LIN {X 0,Y 573.241,Z 599.114,A -85,B 0,C 180,E1 -2241.185,E2 -2241.185} C_VEL
LIN {X 0,Y 573.161,Z 606.962,A -85,B 0,C 180,E1 -2242.071,E2 -2242.071} C_VEL
LIN {X 0,Y 573.072,Z 614.955,A -85,B 0,C 180,E1 -2243.185,E2 -2243.185} C_VEL
LIN {X 0,Y 573.07,Z 621.68,A -85,B 0,C 180,E1 -2244.37,E2 -2244.37} C_VEL
LIN {X 0,Y 573.029,Z 626.372,A -85,B 0,C 180,E1 -2245.428,E2 -2245.428} C_VEL
LIN {X 0,Y 573.022,Z 629.957,A -85,B 0,C 180,E1 -2246.484,E2 -2246.484} C_VEL
LIN {X 0,Y 572.959,Z 631.808,A -85,B 0,C 180,E1 -2247.188,E2 -2247.188} C_VEL
LIN {X 0,Y 572.938,Z 633.198,A -85,B 0,C 180,E1 -2247.891,E2 -2247.891} C_VEL
LIN {X 0,Y 572.941,Z 634.785,A -85,B 0,C 180,E1 -2249.297,E2 -2249.297} C_VEL
LIN {X 0,Y 572.938,Z 635,A -85,B 0,C 180,E1 -2250,E2 -2250} C_VEL
LIN {X 0,Y 572.946,Z 634.186,A -85,B 0,C 180,E1 -2251.406,E2 -2251.406} C_VEL
LIN {X 0,Y 572.938,Z 633.2,A -85,B 0,C 180,E1 -2252.109,E2 -2252.109} C_VEL
LIN {X 0,Y 572.959,Z 631.81,A -85,B 0,C 180,E1 -2252.812,E2 -2252.812} C_VEL
LIN {X 0,Y 573.014,Z 628.896,A -85,B 0,C 180,E1 -2253.868,E2 -2253.868} C_VEL
LIN {X 0,Y 572.963,Z 624.949,A -85,B 0,C 180,E1 -2254.926,E2 -2254.926} C_VEL
LIN {X 0,Y 573.064,Z 618.877,A -85,B 0,C 180,E1 -2256.16,E2 -2256.16} C_VEL
LIN {X 0,Y 573.119,Z 612.238,A -85,B 0,C 180,E1 -2257.221,E2 -2257.221} C_VEL
LIN {X 0,Y 573.201,Z 603.992,A -85,B 0,C 180,E1 -2258.283,E2 -2258.283} C_VEL
LIN {X 0,Y 573.286,Z 595.54,A -85,B 0,C 180,E1 -2259.17,E2 -2259.17} C_VEL
LIN {X 0,Y 573.421,Z 585.101,A -85,B 0,C 180,E1 -2260.058,E2 -2260.058} C_VEL
LIN {X 0,Y 573.55,Z 573.355,A -85,B 0,C 180,E1 -2260.858,E2 -2260.858} C_VEL
LIN {X 0,Y 573.653,Z 562.287,A -85,B 0,C 180,E1 -2261.447,E2 -2261.447} C_VEL
LIN {X 0,Y 573.748,Z 549.178,A -85,B 0,C 180,E1 -2261.974,E2 -2261.974} C_VEL
LIN {X 0,Y 573.828,Z 536.528,A -85,B 0,C 180,E1 -2262.331,E2 -2262.331} C_VEL
LIN {X 0,Y 573.892,Z 523.328,A -85,B 0,C 180,E1 -2262.554,E2 -2262.554} C_VEL
LIN {X 0,Y 573.889,Z 423.833,A -85,B 0,C 180,E1 -2263.807,E2 -2263.807} C_VEL
LIN {X 0,Y 573.519,Z 420.897,A -85,B 0,C 180,E1 -2263.87,E2 -2263.87} C_VEL
LIN {X 0,Y 573.775,Z 395.95,A -85,B 0,C 180,E1 -2266.546,E2 -2266.546} C_VEL
LIN {X 0,Y 574.061,Z 369.009,A -85,B 0,C 180,E1 -2269.493,E2 -2269.493} C_VEL
LIN {X 0,Y 574.387,Z 343.84,A -85,B 0,C 180,E1 -2272.29,E2 -2272.29} C_VEL
LIN {X 0,Y 574.532,Z 322.946,A -85,B 0,C 180,E1 -2274.576,E2 -2274.576} C_VEL
LIN {X 0,Y 574.612,Z 306.194,A -85,B 0,C 180,E1 -2276.412,E2 -2276.412} C_VEL
LIN {X 0,Y 573.247,Z 300.208,A -85,B 0,C 180,E1 -2277.16,E2 -2277.16} C_VEL
LIN {X 0,Y 573.225,Z 300.08,A -85,B 0,C 180,E1 -2280.177,E2 -2280.177} C_VEL
LIN {X 0,Y 573.221,Z 300.078,A -85,B 0,C 180,E1 -2282.646,E2 -2282.646} C_VEL
LIN {X 0,Y 573.184,Z 300.082,A -85,B 0,C 180,E1 -2285.189,E2 -2285.189} C_VEL
LIN {X 0,Y 573.216,Z 300.084,A -85,B 0,C 180,E1 -2287.808,E2 -2287.808} C_VEL
LIN {X 0,Y 573.242,Z 300.076,A -85,B 0,C 180,E1 -2290.524,E2 -2290.524} C_VEL
LIN {X 0,Y 573.199,Z 300.084,A -85,B 0,C 180,E1 -2293.664,E2 -2293.664} C_VEL
LIN {X 0,Y 573.195,Z 300.08,A -85,B 0,C 180,E1 -2296.637,E2 -2296.637} C_VEL
LIN {X 0,Y 573.24,Z 300.077,A -85,B 0,C 180,E1 -2299.474,E2 -2299.474} C_VEL
LIN {X 0,Y 573.212,Z 300.075,A -85,B 0,C 180,E1 -2302.19,E2 -2302.19} C_VEL
LIN {X 0,Y 573.213,Z 300.075,A -85,B 0,C 180,E1 -2305.23,E2 -2305.23} C_VEL
LIN {X 0,Y 573.241,Z 300.082,A -85,B 0,C 180,E1 -2307.772,E2 -2307.772} C_VEL
LIN {X 0,Y 573.253,Z 300.071,A -85,B 0,C 180,E1 -2310.633,E2 -2310.633} C_VEL
LIN {X 0,Y 573.198,Z 300.083,A -85,B 0,C 180,E1 -2313.513,E2 -2313.513} C_VEL
LIN {X 0,Y 573.21,Z 300.082,A -85,B 0,C 180,E1 -2316.134,E2 -2316.134} C_VEL
LIN {X 0,Y 573.239,Z 300.072,A -85,B 0,C 180,E1 -2319.173,E2 -2319.173} C_VEL
LIN {X 0,Y 573.199,Z 300.081,A -85,B 0,C 180,E1 -2321.41,E2 -2321.41} C_VEL
LIN {X 0,Y 573.227,Z 300.083,A -85,B 0,C 180,E1 -2323.621,E2 -2323.621} C_VEL
LIN {X 0,Y 573.253,Z 300.08,A -85,B 0,C 180,E1 -2325.806,E2 -2325.806} C_VEL
LIN {X 0,Y 573.254,Z 300.072,A -85,B 0,C 180,E1 -2328.745,E2 -2328.745} C_VEL
LIN {X 0,Y 573.231,Z 300.082,A -85,B 0,C 180,E1 -2331.54,E2 -2331.54} C_VEL
LIN {X 0,Y 573.224,Z 300.084,A -85,B 0,C 180,E1 -2333.665,E2 -2333.665} C_VEL
LIN {X 0,Y 573.203,Z 300.088,A -85,B 0,C 180,E1 -2335.781,E2 -2335.781} C_VEL
LIN {X 0,Y 573.287,Z 300.075,A -85,B 0,C 180,E1 -2337.892,E2 -2337.892} C_VEL
LIN {X 0,Y 573.298,Z 300.069,A -85,B 0,C 180,E1 -2340,E2 -2340} C_VEL
LIN {X 0,Y 573.272,Z 300.069,A -85,B 0,C 180,E1 -2342.811,E2 -2342.811} C_VEL
LIN {X 0,Y 573.268,Z 300.08,A -85,B 0,C 180,E1 -2345.628,E2 -2345.628} C_VEL
LIN {X 0,Y 573.233,Z 300.073,A -85,B 0,C 180,E1 -2348.46,E2 -2348.46} C_VEL
LIN {X 0,Y 573.263,Z 300.076,A -85,B 0,C 180,E1 -2351.312,E2 -2351.312} C_VEL
LIN {X 0,Y 573.248,Z 300.071,A -85,B 0,C 180,E1 -2354.415,E2 -2354.415} C_VEL
LIN {X 0,Y 573.228,Z 300.078,A -85,B 0,C 180,E1 -2357.113,E2 -2357.113} C_VEL
LIN {X 0,Y 573.221,Z 300.077,A -85,B 0,C 180,E1 -2360.078,E2 -2360.078} C_VEL
LIN {X 0,Y 573.21,Z 300.078,A -85,B 0,C 180,E1 -2362.339,E2 -2362.339} C_VEL
LIN {X 0,Y 573.188,Z 300.081,A -85,B 0,C 180,E1 -2364.345,E2 -2364.345} C_VEL
LIN {X 0,Y 572.549,Z 300.162,A -85,B 0,C 180,E1 -2364.932,E2 -2364.932} C_VEL
LIN {X 0,Y 569.716,Z 300.521,A -85,B 0,C 180,E1 -2365.883,E2 -2365.883} C_VEL
LIN {X 0,Y 567.297,Z 300.825,A -85,B 0,C 180,E1 -2366.649,E2 -2366.649} C_VEL
LIN {X 0,Y 566.241,Z 300.953,A -85,B 0,C 180,E1 -2367.24,E2 -2367.24} C_VEL
LIN {X 0,Y 566.147,Z 300.961,A -85,B 0,C 180,E1 -2367.441,E2 -2367.441} C_VEL
LIN {X 0,Y 566.16,Z 300.956,A -85,B 0,C 180,E1 -2369.771,E2 -2369.771} C_VEL
LIN {X 0,Y 566.184,Z 300.951,A -85,B 0,C 180,E1 -2372.428,E2 -2372.428} C_VEL
LIN {X 0,Y 566.159,Z 300.959,A -85,B 0,C 180,E1 -2374.988,E2 -2374.988} C_VEL
LIN {X 0,Y 566.182,Z 300.959,A -85,B 0,C 180,E1 -2377.462,E2 -2377.462} C_VEL
LIN {X 0,Y 566.188,Z 300.95,A -85,B 0,C 180,E1 -2380.201,E2 -2380.201} C_VEL
LIN {X 0,Y 566.175,Z 300.958,A -85,B 0,C 180,E1 -2383.057,E2 -2383.057} C_VEL
LIN {X 0,Y 566.149,Z 300.955,A -85,B 0,C 180,E1 -2386.054,E2 -2386.054} C_VEL
LIN {X 0,Y 566.149,Z 300.959,A -85,B 0,C 180,E1 -2388.859,E2 -2388.859} C_VEL
LIN {X 0,Y 566.195,Z 300.958,A -85,B 0,C 180,E1 -2391.444,E2 -2391.444} C_VEL
LIN {X 0,Y 566.139,Z 300.958,A -85,B 0,C 180,E1 -2394.307,E2 -2394.307} C_VEL
LIN {X 0,Y 566.165,Z 300.958,A -85,B 0,C 180,E1 -2396.895,E2 -2396.895} C_VEL
LIN {X 0,Y 566.158,Z 300.965,A -85,B 0,C 180,E1 -2399.407,E2 -2399.407} C_VEL
LIN {X 0,Y 566.151,Z 300.954,A -85,B 0,C 180,E1 -2401.855,E2 -2401.855} C_VEL
LIN {X 0,Y 566.169,Z 300.955,A -85,B 0,C 180,E1 -2404.249,E2 -2404.249} C_VEL
LIN {X 0,Y 566.159,Z 300.961,A -85,B 0,C 180,E1 -2407.368,E2 -2407.368} C_VEL
LIN {X 0,Y 566.199,Z 300.956,A -85,B 0,C 180,E1 -2409.663,E2 -2409.663} C_VEL
LIN {X 0,Y 566.196,Z 300.944,A -85,B 0,C 180,E1 -2412.897,E2 -2412.897} C_VEL
LIN {X 0,Y 566.221,Z 300.986,A -85,B 0,C 180,E1 -2416.222,E2 -2416.222} C_VEL
LIN {X 0,Y 566.335,Z 301.687,A -85,B 0,C 180,E1 -2416.374,E2 -2416.374} C_VEL
LIN {X 0,Y 567.038,Z 303.971,A -85,B 0,C 180,E1 -2416.453,E2 -2416.453} C_VEL
LIN {X 0,Y 566.993,Z 380.985,A -85,B 0,C 180,E1 -2417.45,E2 -2417.45} C_VEL
LIN {X 0,Y 566.878,Z 394.243,A -85,B 0,C 180,E1 -2417.765,E2 -2417.765} C_VEL
LIN {X 0,Y 566.749,Z 406.398,A -85,B 0,C 180,E1 -2418.194,E2 -2418.194} C_VEL
LIN {X 0,Y 566.633,Z 418.541,A -85,B 0,C 180,E1 -2418.775,E2 -2418.775} C_VEL
LIN {X 0,Y 566.473,Z 429.557,A -85,B 0,C 180,E1 -2419.456,E2 -2419.456} C_VEL
LIN {X 0,Y 566.326,Z 440.075,A -85,B 0,C 180,E1 -2420.266,E2 -2420.266} C_VEL
LIN {X 0,Y 566.221,Z 448.673,A -85,B 0,C 180,E1 -2421.075,E2 -2421.075} C_VEL
LIN {X 0,Y 566.113,Z 456.592,A -85,B 0,C 180,E1 -2421.972,E2 -2421.972} C_VEL
LIN {X 0,Y 566.05,Z 463.16,A -85,B 0,C 180,E1 -2422.868,E2 -2422.868} C_VEL
LIN {X 0,Y 566.003,Z 469.628,A -85,B 0,C 180,E1 -2423.942,E2 -2423.942} C_VEL
LIN {X 0,Y 565.878,Z 474.766,A -85,B 0,C 180,E1 -2425.013,E2 -2425.013} C_VEL
LIN {X 0,Y 565.926,Z 478.754,A -85,B 0,C 180,E1 -2426.084,E2 -2426.084} C_VEL
LIN {X 0,Y 565.877,Z 481.704,A -85,B 0,C 180,E1 -2427.153,E2 -2427.153} C_VEL
LIN {X 0,Y 565.84,Z 483.127,A -85,B 0,C 180,E1 -2427.865,E2 -2427.865} C_VEL
LIN {X 0,Y 565.841,Z 484.756,A -85,B 0,C 180,E1 -2429.288,E2 -2429.288} C_VEL
LIN {X 0,Y 565.839,Z 484.996,A -85,B 0,C 180,E1 -2430,E2 -2430} C_VEL
LIN {X 0,Y 565.841,Z 484.815,A -85,B 0,C 180,E1 -2430.712,E2 -2430.712} C_VEL
LIN {X 0,Y 565.841,Z 483.269,A -85,B 0,C 180,E1 -2432.135,E2 -2432.135} C_VEL
LIN {X 0,Y 565.878,Z 481.908,A -85,B 0,C 180,E1 -2432.847,E2 -2432.847} C_VEL
LIN {X 0,Y 565.927,Z 479.029,A -85,B 0,C 180,E1 -2433.916,E2 -2433.916} C_VEL
LIN {X 0,Y 565.878,Z 475.129,A -85,B 0,C 180,E1 -2434.987,E2 -2434.987} C_VEL
LIN {X 0,Y 565.99,Z 470.098,A -85,B 0,C 180,E1 -2436.059,E2 -2436.059} C_VEL
LIN {X 0,Y 566.031,Z 463.773,A -85,B 0,C 180,E1 -2437.132,E2 -2437.132} C_VEL
LIN {X 0,Y 566.128,Z 455.85,A -85,B 0,C 180,E1 -2438.208,E2 -2438.208} C_VEL
LIN {X 0,Y 566.249,Z 445.997,A -85,B 0,C 180,E1 -2439.285,E2 -2439.285} C_VEL
LIN {X 0,Y 566.425,Z 435.682,A -85,B 0,C 180,E1 -2440.184,E2 -2440.184} C_VEL
LIN {X 0,Y 566.581,Z 424.398,A -85,B 0,C 180,E1 -2440.971,E2 -2440.971} C_VEL
LIN {X 0,Y 566.679,Z 412.486,A -85,B 0,C 180,E1 -2441.626,E2 -2441.626} C_VEL
LIN {X 0,Y 566.819,Z 400.474,A -85,B 0,C 180,E1 -2442.123,E2 -2442.123} C_VEL
LIN {X 0,Y 566.928,Z 387.43,A -85,B 0,C 180,E1 -2442.506,E2 -2442.506} C_VEL
LIN {X 0,Y 567.026,Z 375.066,A -85,B 0,C 180,E1 -2442.732,E2 -2442.732} C_VEL
LIN {X 0,Y 567.08,Z 304.212,A -85,B 0,C 180,E1 -2443.633,E2 -2443.633} C_VEL
LIN {X 0,Y 566.353,Z 301.818,A -85,B 0,C 180,E1 -2443.706,E2 -2443.706} C_VEL
LIN {X 0,Y 566.205,Z 301.005,A -85,B 0,C 180,E1 -2443.847,E2 -2443.847} C_VEL
LIN {X 0,Y 566.195,Z 300.93,A -85,B 0,C 180,E1 -2447.102,E2 -2447.102} C_VEL
LIN {X 0,Y 566.172,Z 300.956,A -85,B 0,C 180,E1 -2449.582,E2 -2449.582} C_VEL
LIN {X 0,Y 566.181,Z 300.952,A -85,B 0,C 180,E1 -2451.863,E2 -2451.863} C_VEL
LIN {X 0,Y 566.146,Z 300.959,A -85,B 0,C 180,E1 -2454.183,E2 -2454.183} C_VEL
LIN {X 0,Y 566.162,Z 300.961,A -85,B 0,C 180,E1 -2456.649,E2 -2456.649} C_VEL
LIN {X 0,Y 566.154,Z 300.957,A -85,B 0,C 180,E1 -2459.771,E2 -2459.771} C_VEL
LIN {X 0,Y 566.175,Z 300.959,A -85,B 0,C 180,E1 -2462.425,E2 -2462.425} C_VEL
LIN {X 0,Y 566.165,Z 300.961,A -85,B 0,C 180,E1 -2464.987,E2 -2464.987} C_VEL
LIN {X 0,Y 566.18,Z 300.952,A -85,B 0,C 180,E1 -2467.461,E2 -2467.461} C_VEL
LIN {X 0,Y 566.2,Z 300.954,A -85,B 0,C 180,E1 -2470.199,E2 -2470.199} C_VEL
LIN {X 0,Y 566.142,Z 300.959,A -85,B 0,C 180,E1 -2473.059,E2 -2473.059} C_VEL
LIN {X 0,Y 566.14,Z 300.96,A -85,B 0,C 180,E1 -2476.054,E2 -2476.054} C_VEL
LIN {X 0,Y 566.156,Z 300.955,A -85,B 0,C 180,E1 -2479.219,E2 -2479.219} C_VEL
LIN {X 0,Y 566.164,Z 300.951,A -85,B 0,C 180,E1 -2481.635,E2 -2481.635} C_VEL
LIN {X 0,Y 566.132,Z 300.964,A -85,B 0,C 180,E1 -2484.305,E2 -2484.305} C_VEL
LIN {X 0,Y 566.187,Z 300.956,A -85,B 0,C 180,E1 -2486.895,E2 -2486.895} C_VEL
LIN {X 0,Y 566.146,Z 300.952,A -85,B 0,C 180,E1 -2489.405,E2 -2489.405} C_VEL
LIN {X 0,Y 566.139,Z 300.954,A -85,B 0,C 180,E1 -2491.853,E2 -2491.853} C_VEL
LIN {X 0,Y 566.184,Z 300.957,A -85,B 0,C 180,E1 -2494.249,E2 -2494.249} C_VEL
LIN {X 0,Y 566.13,Z 300.959,A -85,B 0,C 180,E1 -2497.366,E2 -2497.366} C_VEL
LIN {X 0,Y 566.161,Z 300.954,A -85,B 0,C 180,E1 -2499.661,E2 -2499.661} C_VEL
LIN {X 0,Y 566.161,Z 300.958,A -85,B 0,C 180,E1 -2501.92,E2 -2501.92} C_VEL
LIN {X 0,Y 566.17,Z 300.955,A -85,B 0,C 180,E1 -2504.89,E2 -2504.89} C_VEL
LIN {X 0,Y 566.163,Z 300.957,A -85,B 0,C 180,E1 -2507.817,E2 -2507.817} C_VEL
LIN {X 0,Y 566.143,Z 300.961,A -85,B 0,C 180,E1 -2509.991,E2 -2509.991} C_VEL
LIN {X 0,Y 566.176,Z 300.956,A -85,B 0,C 180,E1 -2512.869,E2 -2512.869} C_VEL
LIN {X 0,Y 566.245,Z 300.947,A -85,B 0,C 180,E1 -2515.016,E2 -2515.016} C_VEL
LIN {X 0,Y 566.254,Z 300.946,A -85,B 0,C 180,E1 -2517.866,E2 -2517.866} C_VEL
LIN {X 0,Y 566.289,Z 300.944,A -85,B 0,C 180,E1 -2520.711,E2 -2520.711} C_VEL
LIN {X 0,Y 566.247,Z 300.947,A -85,B 0,C 180,E1 -2522.846,E2 -2522.846} C_VEL
LIN {X 0,Y 566.224,Z 300.948,A -85,B 0,C 180,E1 -2525.699,E2 -2525.699} C_VEL
LIN {X 0,Y 566.174,Z 300.956,A -85,B 0,C 180,E1 -2527.848,E2 -2527.848} C_VEL
LIN {X 0,Y 566.204,Z 300.953,A -85,B 0,C 180,E1 -2530.73,E2 -2530.73} C_VEL
LIN {X 0,Y 566.171,Z 300.954,A -85,B 0,C 180,E1 -2533.642,E2 -2533.642} C_VEL
LIN {X 0,Y 566.175,Z 300.958,A -85,B 0,C 180,E1 -2535.848,E2 -2535.848} C_VEL
LIN {X 0,Y 566.18,Z 300.953,A -85,B 0,C 180,E1 -2538.829,E2 -2538.829} C_VEL
LIN {X 0,Y 566.2,Z 300.948,A -85,B 0,C 180,E1 -2541.42,E2 -2541.42} C_VEL
LIN {X 0,Y 566.163,Z 300.965,A -85,B 0,C 180,E1 -2544.182,E2 -2544.182} C_VEL
LIN {X 0,Y 566.166,Z 300.956,A -85,B 0,C 180,E1 -2546.653,E2 -2546.653} C_VEL
LIN {X 0,Y 566.166,Z 300.954,A -85,B 0,C 180,E1 -2548.955,E2 -2548.955} C_VEL
LIN {X 0,Y 566.182,Z 300.954,A -85,B 0,C 180,E1 -2551.423,E2 -2551.423} C_VEL
LIN {X 0,Y 566.188,Z 300.959,A -85,B 0,C 180,E1 -2553.958,E2 -2553.958} C_VEL
LIN {X 0,Y 566.138,Z 300.962,A -85,B 0,C 180,E1 -2556.575,E2 -2556.575} C_VEL
LIN {X 0,Y 566.2,Z 300.95,A -85,B 0,C 180,E1 -2559.275,E2 -2559.275} C_VEL
LIN {X 0,Y 566.173,Z 300.964,A -85,B 0,C 180,E1 -2562.091,E2 -2562.091} C_VEL
LIN {X 0,Y 566.159,Z 300.951,A -85,B 0,C 180,E1 -2565.038,E2 -2565.038} C_VEL
LIN {X 0,Y 566.158,Z 300.964,A -85,B 0,C 180,E1 -2568.143,E2 -2568.143} C_VEL
LIN {X 0,Y 566.204,Z 300.95,A -85,B 0,C 180,E1 -2570.726,E2 -2570.726} C_VEL
LIN {X 0,Y 566.139,Z 300.961,A -85,B 0,C 180,E1 -2573.426,E2 -2573.426} C_VEL
LIN {X 0,Y 566.193,Z 300.956,A -85,B 0,C 180,E1 -2576.269,E2 -2576.269} C_VEL
LIN {X 0,Y 566.181,Z 300.954,A -85,B 0,C 180,E1 -2578.926,E2 -2578.926} C_VEL
LIN {X 0,Y 566.147,Z 300.965,A -85,B 0,C 180,E1 -2581.854,E2 -2581.854} C_VEL
LIN {X 0,Y 566.189,Z 301.12,A -85,B 0,C 180,E1 -2582.681,E2 -2582.681} C_VEL
LIN {X 0,Y 567.751,Z 307.979,A -85,B 0,C 180,E1 -2583.537,E2 -2583.537} C_VEL
LIN {X 0,Y 567.58,Z 332.208,A -85,B 0,C 180,E1 -2586.22,E2 -2586.22} C_VEL
LIN {X 0,Y 567.362,Z 357.278,A -85,B 0,C 180,E1 -2588.948,E2 -2588.948} C_VEL
LIN {X 0,Y 566.967,Z 384.183,A -85,B 0,C 180,E1 -2591.947,E2 -2591.947} C_VEL
LIN {X 0,Y 566.677,Z 409.398,A -85,B 0,C 180,E1 -2594.72,E2 -2594.72} C_VEL
LIN {X 0,Y 566.563,Z 420.903,A -85,B 0,C 180,E1 -2595.956,E2 -2595.956} C_VEL
LIN {X 0,Y 567.197,Z 426.739,A -85,B 0,C 180,E1 -2596.064,E2 -2596.064} C_VEL
LIN {X 0,Y 566.97,Z 530.957,A -85,B 0,C 180,E1 -2597.404,E2 -2597.404} C_VEL
LIN {X 0,Y 566.892,Z 543.463,A -85,B 0,C 180,E1 -2597.697,E2 -2597.697} C_VEL
LIN {X 0,Y 566.747,Z 555.924,A -85,B 0,C 180,E1 -2598.13,E2 -2598.13} C_VEL
LIN {X 0,Y 566.627,Z 568.166,A -85,B 0,C 180,E1 -2598.709,E2 -2598.709} C_VEL
LIN {X 0,Y 566.457,Z 580.202,A -85,B 0,C 180,E1 -2599.456,E2 -2599.456} C_VEL
LIN {X 0,Y 566.321,Z 590.604,A -85,B 0,C 180,E1 -2600.266,E2 -2600.266} C_VEL
LIN {X 0,Y 566.207,Z 599.114,A -85,B 0,C 180,E1 -2601.074,E2 -2601.074} C_VEL
LIN {X 0,Y 566.112,Z 606.962,A -85,B 0,C 180,E1 -2601.972,E2 -2601.972} C_VEL
LIN {X 0,Y 566.003,Z 614.623,A -85,B 0,C 180,E1 -2603.047,E2 -2603.047} C_VEL
LIN {X 0,Y 566.004,Z 621.68,A -85,B 0,C 180,E1 -2604.299,E2 -2604.299} C_VEL
LIN {X 0,Y 565.933,Z 626.372,A -85,B 0,C 180,E1 -2605.37,E2 -2605.37} C_VEL
LIN {X 0,Y 565.927,Z 629.958,A -85,B 0,C 180,E1 -2606.44,E2 -2606.44} C_VEL
LIN {X 0,Y 565.878,Z 631.808,A -85,B 0,C 180,E1 -2607.152,E2 -2607.152} C_VEL
LIN {X 0,Y 565.846,Z 634.185,A -85,B 0,C 180,E1 -2608.577,E2 -2608.577} C_VEL
LIN {X 0,Y 565.839,Z 635,A -85,B 0,C 180,E1 -2610,E2 -2610} C_VEL
LIN {X 0,Y 565.846,Z 634.186,A -85,B 0,C 180,E1 -2611.423,E2 -2611.423} C_VEL
LIN {X 0,Y 565.878,Z 631.81,A -85,B 0,C 180,E1 -2612.847,E2 -2612.847} C_VEL
LIN {X 0,Y 565.926,Z 628.896,A -85,B 0,C 180,E1 -2613.916,E2 -2613.916} C_VEL
LIN {X 0,Y 565.878,Z 624.949,A -85,B 0,C 180,E1 -2614.987,E2 -2614.987} C_VEL
LIN {X 0,Y 566.002,Z 619.867,A -85,B 0,C 180,E1 -2616.058,E2 -2616.058} C_VEL
LIN {X 0,Y 566.04,Z 613.469,A -85,B 0,C 180,E1 -2617.132,E2 -2617.132} C_VEL
LIN {X 0,Y 566.133,Z 605.479,A -85,B 0,C 180,E1 -2618.208,E2 -2618.208} C_VEL
LIN {X 0,Y 566.228,Z 597.337,A -85,B 0,C 180,E1 -2619.105,E2 -2619.105} C_VEL
LIN {X 0,Y 566.342,Z 587.402,A -85,B 0,C 180,E1 -2620.005,E2 -2620.005} C_VEL
LIN {X 0,Y 566.525,Z 576.288,A -85,B 0,C 180,E1 -2620.808,E2 -2620.808} C_VEL
LIN {X 0,Y 566.66,Z 565.18,A -85,B 0,C 180,E1 -2621.446,E2 -2621.446} C_VEL
LIN {X 0,Y 566.737,Z 552.988,A -85,B 0,C 180,E1 -2621.988,E2 -2621.988} C_VEL
LIN {X 0,Y 566.906,Z 540.185,A -85,B 0,C 180,E1 -2622.393,E2 -2622.393} C_VEL
LIN {X 0,Y 566.995,Z 526.617,A -85,B 0,C 180,E1 -2622.664,E2 -2622.664} C_VEL
LIN {X 0,Y 567.067,Z 424.95,A -85,B 0,C 180,E1 -2623.962,E2 -2623.962} C_VEL
LIN {X 0,Y 566.562,Z 420.904,A -85,B 0,C 180,E1 -2624.044,E2 -2624.044} C_VEL
LIN {X 0,Y 566.844,Z 394.447,A -85,B 0,C 180,E1 -2626.92,E2 -2626.92} C_VEL
LIN {X 0,Y 567.215,Z 367.71,A -85,B 0,C 180,E1 -2629.884,E2 -2629.884} C_VEL
LIN {X 0,Y 567.445,Z 346.786,A -85,B 0,C 180,E1 -2632.194,E2 -2632.194} C_VEL
LIN {X 0,Y 567.647,Z 322.094,A -85,B 0,C 180,E1 -2634.894,E2 -2634.894} C_VEL
LIN {X 0,Y 567.737,Z 307.968,A -85,B 0,C 180,E1 -2636.464,E2 -2636.464} C_VEL
LIN {X 0,Y 566.207,Z 301.1,A -85,B 0,C 180,E1 -2637.32,E2 -2637.32} C_VEL
LIN {X 0,Y 566.158,Z 300.954,A -85,B 0,C 180,E1 -2639.771,E2 -2639.771} C_VEL
LIN {X 0,Y 566.176,Z 300.958,A -85,B 0,C 180,E1 -2642.425,E2 -2642.425} C_VEL
LIN {X 0,Y 566.16,Z 300.956,A -85,B 0,C 180,E1 -2644.986,E2 -2644.986} C_VEL
LIN {X 0,Y 566.182,Z 300.956,A -85,B 0,C 180,E1 -2647.461,E2 -2647.461} C_VEL
LIN {X 0,Y 566.202,Z 300.957,A -85,B 0,C 180,E1 -2650.199,E2 -2650.199} C_VEL
LIN {X 0,Y 566.143,Z 300.958,A -85,B 0,C 180,E1 -2653.059,E2 -2653.059} C_VEL
LIN {X 0,Y 566.152,Z 300.964,A -85,B 0,C 180,E1 -2656.053,E2 -2656.053} C_VEL
LIN {X 0,Y 566.151,Z 300.957,A -85,B 0,C 180,E1 -2658.858,E2 -2658.858} C_VEL
LIN {X 0,Y 566.195,Z 300.952,A -85,B 0,C 180,E1 -2661.443,E2 -2661.443} C_VEL
LIN {X 0,Y 566.133,Z 300.959,A -85,B 0,C 180,E1 -2664.306,E2 -2664.306} C_VEL
LIN {X 0,Y 566.191,Z 300.952,A -85,B 0,C 180,E1 -2666.896,E2 -2666.896} C_VEL
LIN {X 0,Y 566.174,Z 300.957,A -85,B 0,C 180,E1 -2669.407,E2 -2669.407} C_VEL
LIN {X 0,Y 566.18,Z 300.96,A -85,B 0,C 180,E1 -2671.856,E2 -2671.856} C_VEL
LIN {X 0,Y 566.179,Z 300.957,A -85,B 0,C 180,E1 -2674.249,E2 -2674.249} C_VEL
LIN {X 0,Y 566.157,Z 300.956,A -85,B 0,C 180,E1 -2676.72,E2 -2676.72} C_VEL
LIN {X 0,Y 566.195,Z 300.955,A -85,B 0,C 180,E1 -2679.662,E2 -2679.662} C_VEL
LIN {X 0,Y 566.169,Z 300.963,A -85,B 0,C 180,E1 -2681.921,E2 -2681.921} C_VEL
LIN {X 0,Y 566.18,Z 300.957,A -85,B 0,C 180,E1 -2684.152,E2 -2684.152} C_VEL
LIN {X 0,Y 566.171,Z 300.954,A -85,B 0,C 180,E1 -2686.358,E2 -2686.358} C_VEL
LIN {X 0,Y 566.222,Z 300.95,A -85,B 0,C 180,E1 -2689.27,E2 -2689.27} C_VEL
LIN {X 0,Y 566.175,Z 300.956,A -85,B 0,C 180,E1 -2692.152,E2 -2692.152} C_VEL
LIN {X 0,Y 566.226,Z 300.948,A -85,B 0,C 180,E1 -2694.301,E2 -2694.301} C_VEL
LIN {X 0,Y 566.248,Z 300.947,A -85,B 0,C 180,E1 -2697.154,E2 -2697.154} C_VEL
LIN {X 0,Y 566.268,Z 300.945,A -85,B 0,C 180,E1 -2700,E2 -2700} C_VEL
LIN {X 0,Y 566.242,Z 300.945,A -85,B 0,C 180,E1 -2702.846,E2 -2702.846} C_VEL
LIN {X 0,Y 566.235,Z 300.955,A -85,B 0,C 180,E1 -2705.699,E2 -2705.699} C_VEL
LIN {X 0,Y 566.185,Z 300.951,A -85,B 0,C 180,E1 -2708.566,E2 -2708.566} C_VEL
LIN {X 0,Y 566.23,Z 300.954,A -85,B 0,C 180,E1 -2711.455,E2 -2711.455} C_VEL
LIN {X 0,Y 566.204,Z 300.948,A -85,B 0,C 180,E1 -2714.498,E2 -2714.498} C_VEL
LIN {X 0,Y 566.173,Z 300.96,A -85,B 0,C 180,E1 -2717.333,E2 -2717.333} C_VEL
LIN {X 0,Y 566.19,Z 300.961,A -85,B 0,C 180,E1 -2719.582,E2 -2719.582} C_VEL
LIN {X 0,Y 566.176,Z 300.958,A -85,B 0,C 180,E1 -2721.863,E2 -2721.863} C_VEL
LIN {X 0,Y 566.17,Z 300.957,A -85,B 0,C 180,E1 -2725.022,E2 -2725.022} C_VEL
LIN {X 0,Y 566.147,Z 300.961,A -85,B 0,C 180,E1 -2727.441,E2 -2727.441} C_VEL
LIN {X 0,Y 565.459,Z 301.041,A -85,B 0,C 180,E1 -2728.034,E2 -2728.034} C_VEL
LIN {X 0,Y 562.605,Z 301.395,A -85,B 0,C 180,E1 -2728.999,E2 -2728.999} C_VEL
LIN {X 0,Y 560.214,Z 301.696,A -85,B 0,C 180,E1 -2729.775,E2 -2729.775} C_VEL
LIN {X 0,Y 559.197,Z 301.817,A -85,B 0,C 180,E1 -2730.373,E2 -2730.373} C_VEL
LIN {X 0,Y 559.118,Z 301.827,A -85,B 0,C 180,E1 -2730.576,E2 -2730.576} C_VEL
LIN {X 0,Y 559.14,Z 301.829,A -85,B 0,C 180,E1 -2732.717,E2 -2732.717} C_VEL
LIN {X 0,Y 559.109,Z 301.842,A -85,B 0,C 180,E1 -2735.326,E2 -2735.326} C_VEL
LIN {X 0,Y 559.116,Z 301.831,A -85,B 0,C 180,E1 -2738.019,E2 -2738.019} C_VEL
LIN {X 0,Y 559.143,Z 301.829,A -85,B 0,C 180,E1 -2739.941,E2 -2739.941} C_VEL
LIN {X 0,Y 559.12,Z 301.839,A -85,B 0,C 180,E1 -2743.195,E2 -2743.195} C_VEL
LIN {X 0,Y 559.116,Z 301.834,A -85,B 0,C 180,E1 -2745.765,E2 -2745.765} C_VEL
LIN {X 0,Y 559.096,Z 301.835,A -85,B 0,C 180,E1 -2748.225,E2 -2748.225} C_VEL
LIN {X 0,Y 559.163,Z 301.833,A -85,B 0,C 180,E1 -2751.066,E2 -2751.066} C_VEL
LIN {X 0,Y 559.113,Z 301.837,A -85,B 0,C 180,E1 -2753.788,E2 -2753.788} C_VEL
LIN {X 0,Y 559.123,Z 301.832,A -85,B 0,C 180,E1 -2756.423,E2 -2756.423} C_VEL
LIN {X 0,Y 559.142,Z 301.834,A -85,B 0,C 180,E1 -2758.98,E2 -2758.98} C_VEL
LIN {X 0,Y 559.111,Z 301.833,A -85,B 0,C 180,E1 -2761.63,E2 -2761.63} C_VEL
LIN {X 0,Y 559.14,Z 301.832,A -85,B 0,C 180,E1 -2763.901,E2 -2763.901} C_VEL
LIN {X 0,Y 559.11,Z 301.841,A -85,B 0,C 180,E1 -2767.067,E2 -2767.067} C_VEL
LIN {X 0,Y 559.171,Z 301.835,A -85,B 0,C 180,E1 -2769.396,E2 -2769.396} C_VEL
LIN {X 0,Y 559.122,Z 301.822,A -85,B 0,C 180,E1 -2772.442,E2 -2772.442} C_VEL
LIN {X 0,Y 559.154,Z 301.835,A -85,B 0,C 180,E1 -2775.441,E2 -2775.441} C_VEL
LIN {X 0,Y 559.229,Z 302.09,A -85,B 0,C 180,E1 -2776.14,E2 -2776.14} C_VEL
LIN {X 0,Y 559.536,Z 303.423,A -85,B 0,C 180,E1 -2776.248,E2 -2776.248} C_VEL
LIN {X 0,Y 560.273,Z 305.992,A -85,B 0,C 180,E1 -2776.305,E2 -2776.305} C_VEL
LIN {X 0,Y 560.089,Z 381.28,A -85,B 0,C 180,E1 -2777.292,E2 -2777.292} C_VEL
LIN {X 0,Y 559.939,Z 394.48,A -85,B 0,C 180,E1 -2777.611,E2 -2777.611} C_VEL
LIN {X 0,Y 559.798,Z 406.547,A -85,B 0,C 180,E1 -2778.045,E2 -2778.045} C_VEL
LIN {X 0,Y 559.648,Z 418.106,A -85,B 0,C 180,E1 -2778.607,E2 -2778.607} C_VEL
LIN {X 0,Y 559.489,Z 429.562,A -85,B 0,C 180,E1 -2779.323,E2 -2779.323} C_VEL
LIN {X 0,Y 559.307,Z 440.08,A -85,B 0,C 180,E1 -2780.142,E2 -2780.142} C_VEL
LIN {X 0,Y 559.197,Z 448.678,A -85,B 0,C 180,E1 -2780.962,E2 -2780.962} C_VEL
LIN {X 0,Y 559.05,Z 456.597,A -85,B 0,C 180,E1 -2781.87,E2 -2781.87} C_VEL
LIN {X 0,Y 558.971,Z 464.457,A -85,B 0,C 180,E1 -2782.977,E2 -2782.977} C_VEL
LIN {X 0,Y 558.936,Z 471.455,A -85,B 0,C 180,E1 -2784.227,E2 -2784.227} C_VEL
LIN {X 0,Y 558.827,Z 476.197,A -85,B 0,C 180,E1 -2785.311,E2 -2785.311} C_VEL
LIN {X 0,Y 558.836,Z 479.828,A -85,B 0,C 180,E1 -2786.395,E2 -2786.395} C_VEL
LIN {X 0,Y 558.799,Z 481.706,A -85,B 0,C 180,E1 -2787.116,E2 -2787.116} C_VEL
LIN {X 0,Y 558.746,Z 483.128,A -85,B 0,C 180,E1 -2787.838,E2 -2787.838} C_VEL
LIN {X 0,Y 558.741,Z 484.756,A -85,B 0,C 180,E1 -2789.279,E2 -2789.279} C_VEL
LIN {X 0,Y 558.74,Z 484.996,A -85,B 0,C 180,E1 -2790,E2 -2790} C_VEL
LIN {X 0,Y 558.741,Z 484.815,A -85,B 0,C 180,E1 -2790.721,E2 -2790.721} C_VEL
LIN {X 0,Y 558.746,Z 483.268,A -85,B 0,C 180,E1 -2792.163,E2 -2792.163} C_VEL
LIN {X 0,Y 558.8,Z 481.907,A -85,B 0,C 180,E1 -2792.884,E2 -2792.884} C_VEL
LIN {X 0,Y 558.844,Z 479.027,A -85,B 0,C 180,E1 -2793.966,E2 -2793.966} C_VEL
LIN {X 0,Y 558.798,Z 475.127,A -85,B 0,C 180,E1 -2795.051,E2 -2795.051} C_VEL
LIN {X 0,Y 558.91,Z 470.095,A -85,B 0,C 180,E1 -2796.136,E2 -2796.136} C_VEL
LIN {X 0,Y 558.972,Z 463.769,A -85,B 0,C 180,E1 -2797.223,E2 -2797.223} C_VEL
LIN {X 0,Y 559.091,Z 455.845,A -85,B 0,C 180,E1 -2798.312,E2 -2798.312} C_VEL
LIN {X 0,Y 559.182,Z 447.774,A -85,B 0,C 180,E1 -2799.221,E2 -2799.221} C_VEL
LIN {X 0,Y 559.357,Z 437.924,A -85,B 0,C 180,E1 -2800.131,E2 -2800.131} C_VEL
LIN {X 0,Y 559.581,Z 427.089,A -85,B 0,C 180,E1 -2800.937,E2 -2800.937} C_VEL
LIN {X 0,Y 559.68,Z 415.301,A -85,B 0,C 180,E1 -2801.631,E2 -2801.631} C_VEL
LIN {X 0,Y 559.832,Z 403.126,A -85,B 0,C 180,E1 -2802.184,E2 -2802.184} C_VEL
LIN {X 0,Y 559.976,Z 390.397,A -85,B 0,C 180,E1 -2802.595,E2 -2802.595} C_VEL
LIN {X 0,Y 560.135,Z 378.322,A -85,B 0,C 180,E1 -2802.845,E2 -2802.845} C_VEL
LIN {X 0,Y 560.265,Z 305.8,A -85,B 0,C 180,E1 -2803.788,E2 -2803.788} C_VEL
LIN {X 0,Y 559.318,Z 302.662,A -85,B 0,C 180,E1 -2803.88,E2 -2803.88} C_VEL
LIN {X 0,Y 559.165,Z 301.88,A -85,B 0,C 180,E1 -2804.021,E2 -2804.021} C_VEL
LIN {X 0,Y 559.149,Z 301.804,A -85,B 0,C 180,E1 -2807.204,E2 -2807.204} C_VEL
LIN {X 0,Y 559.138,Z 301.832,A -85,B 0,C 180,E1 -2809.838,E2 -2809.838} C_VEL
LIN {X 0,Y 559.125,Z 301.832,A -85,B 0,C 180,E1 -2812.153,E2 -2812.153} C_VEL
LIN {X 0,Y 559.115,Z 301.837,A -85,B 0,C 180,E1 -2815.172,E2 -2815.172} C_VEL
LIN {X 0,Y 559.102,Z 301.829,A -85,B 0,C 180,E1 -2817.716,E2 -2817.716} C_VEL
LIN {X 0,Y 559.098,Z 301.837,A -85,B 0,C 180,E1 -2820.185,E2 -2820.185} C_VEL
LIN {X 0,Y 559.133,Z 301.839,A -85,B 0,C 180,E1 -2822.716,E2 -2822.716} C_VEL
LIN {X 0,Y 559.115,Z 301.835,A -85,B 0,C 180,E1 -2825.324,E2 -2825.324} C_VEL
LIN {X 0,Y 559.117,Z 301.832,A -85,B 0,C 180,E1 -2828.018,E2 -2828.018} C_VEL
LIN {X 0,Y 559.12,Z 301.84,A -85,B 0,C 180,E1 -2830.815,E2 -2830.815} C_VEL
LIN {X 0,Y 559.094,Z 301.832,A -85,B 0,C 180,E1 -2833.738,E2 -2833.738} C_VEL
LIN {X 0,Y 559.088,Z 301.841,A -85,B 0,C 180,E1 -2836.261,E2 -2836.261} C_VEL
LIN {X 0,Y 559.109,Z 301.833,A -85,B 0,C 180,E1 -2839.183,E2 -2839.183} C_VEL
LIN {X 0,Y 559.137,Z 301.828,A -85,B 0,C 180,E1 -2841.195,E2 -2841.195} C_VEL
LIN {X 0,Y 559.109,Z 301.834,A -85,B 0,C 180,E1 -2843.787,E2 -2843.787} C_VEL
LIN {X 0,Y 559.138,Z 301.838,A -85,B 0,C 180,E1 -2846.423,E2 -2846.423} C_VEL
LIN {X 0,Y 559.133,Z 301.828,A -85,B 0,C 180,E1 -2848.979,E2 -2848.979} C_VEL
LIN {X 0,Y 559.1,Z 301.829,A -85,B 0,C 180,E1 -2851.63,E2 -2851.63} C_VEL
LIN {X 0,Y 559.15,Z 301.829,A -85,B 0,C 180,E1 -2853.901,E2 -2853.901} C_VEL
LIN {X 0,Y 559.088,Z 301.838,A -85,B 0,C 180,E1 -2857.065,E2 -2857.065} C_VEL
LIN {X 0,Y 559.139,Z 301.828,A -85,B 0,C 180,E1 -2859.394,E2 -2859.394} C_VEL
LIN {X 0,Y 559.11,Z 301.835,A -85,B 0,C 180,E1 -2861.684,E2 -2861.684} C_VEL
LIN {X 0,Y 559.123,Z 301.835,A -85,B 0,C 180,E1 -2863.947,E2 -2863.947} C_VEL
LIN {X 0,Y 559.126,Z 301.835,A -85,B 0,C 180,E1 -2866.183,E2 -2866.183} C_VEL
LIN {X 0,Y 559.169,Z 301.828,A -85,B 0,C 180,E1 -2869.133,E2 -2869.133} C_VEL
LIN {X 0,Y 559.165,Z 301.83,A -85,B 0,C 180,E1 -2872.053,E2 -2872.053} C_VEL
LIN {X 0,Y 559.221,Z 301.822,A -85,B 0,C 180,E1 -2874.953,E2 -2874.953} C_VEL
LIN {X 0,Y 559.227,Z 301.821,A -85,B 0,C 180,E1 -2877.839,E2 -2877.839} C_VEL
LIN {X 0,Y 559.259,Z 301.819,A -85,B 0,C 180,E1 -2880.72,E2 -2880.72} C_VEL
LIN {X 0,Y 559.212,Z 301.823,A -85,B 0,C 180,E1 -2882.881,E2 -2882.881} C_VEL
LIN {X 0,Y 559.196,Z 301.823,A -85,B 0,C 180,E1 -2885.771,E2 -2885.771} C_VEL
LIN {X 0,Y 559.147,Z 301.833,A -85,B 0,C 180,E1 -2888.675,E2 -2888.675} C_VEL
LIN {X 0,Y 559.151,Z 301.829,A -85,B 0,C 180,E1 -2891.602,E2 -2891.602} C_VEL
LIN {X 0,Y 559.192,Z 301.828,A -85,B 0,C 180,E1 -2894.596,E2 -2894.596} C_VEL
LIN {X 0,Y 559.113,Z 301.835,A -85,B 0,C 180,E1 -2897.558,E2 -2897.558} C_VEL
LIN {X 0,Y 559.155,Z 301.83,A -85,B 0,C 180,E1 -2899.838,E2 -2899.838} C_VEL
LIN {X 0,Y 559.129,Z 301.837,A -85,B 0,C 180,E1 -2902.153,E2 -2902.153} C_VEL
LIN {X 0,Y 559.13,Z 301.832,A -85,B 0,C 180,E1 -2905.178,E2 -2905.178} C_VEL
LIN {X 0,Y 559.116,Z 301.835,A -85,B 0,C 180,E1 -2907.716,E2 -2907.716} C_VEL
LIN {X 0,Y 559.14,Z 301.839,A -85,B 0,C 180,E1 -2910.184,E2 -2910.184} C_VEL
LIN {X 0,Y 559.144,Z 301.831,A -85,B 0,C 180,E1 -2912.716,E2 -2912.716} C_VEL
LIN {X 0,Y 559.108,Z 301.833,A -85,B 0,C 180,E1 -2915.326,E2 -2915.326} C_VEL
LIN {X 0,Y 559.117,Z 301.842,A -85,B 0,C 180,E1 -2918.019,E2 -2918.019} C_VEL
LIN {X 0,Y 559.12,Z 301.834,A -85,B 0,C 180,E1 -2920.816,E2 -2920.816} C_VEL
LIN {X 0,Y 559.121,Z 301.832,A -85,B 0,C 180,E1 -2923.195,E2 -2923.195} C_VEL
LIN {X 0,Y 559.118,Z 301.832,A -85,B 0,C 180,E1 -2925.765,E2 -2925.765} C_VEL
LIN {X 0,Y 559.113,Z 301.84,A -85,B 0,C 180,E1 -2928.226,E2 -2928.226} C_VEL
LIN {X 0,Y 559.165,Z 301.826,A -85,B 0,C 180,E1 -2931.193,E2 -2931.193} C_VEL
LIN {X 0,Y 559.11,Z 301.842,A -85,B 0,C 180,E1 -2933.788,E2 -2933.788} C_VEL
LIN {X 0,Y 559.134,Z 301.834,A -85,B 0,C 180,E1 -2936.424,E2 -2936.424} C_VEL
LIN {X 0,Y 559.146,Z 301.831,A -85,B 0,C 180,E1 -2938.981,E2 -2938.981} C_VEL
LIN {X 0,Y 559.167,Z 301.838,A -85,B 0,C 180,E1 -2942.389,E2 -2942.389} C_VEL
LIN {X 0,Y 559.201,Z 302.15,A -85,B 0,C 180,E1 -2942.544,E2 -2942.544} C_VEL
LIN {X 0,Y 560.892,Z 310.659,A -85,B 0,C 180,E1 -2943.589,E2 -2943.589} C_VEL
LIN {X 0,Y 560.617,Z 337.102,A -85,B 0,C 180,E1 -2946.546,E2 -2946.546} C_VEL
LIN {X 0,Y 560.315,Z 363.468,A -85,B 0,C 180,E1 -2949.44,E2 -2949.44} C_VEL
LIN {X 0,Y 560.041,Z 385.864,A -85,B 0,C 180,E1 -2951.906,E2 -2951.906} C_VEL
LIN {X 0,Y 559.682,Z 412.761,A -85,B 0,C 180,E1 -2954.897,E2 -2954.897} C_VEL
LIN {X 0,Y 559.604,Z 420.908,A -85,B 0,C 180,E1 -2955.778,E2 -2955.778} C_VEL
LIN {X 0,Y 560.309,Z 428.527,A -85,B 0,C 180,E1 -2955.912,E2 -2955.912} C_VEL
LIN {X 0,Y 560.047,Z 530.957,A -85,B 0,C 180,E1 -2957.245,E2 -2957.245} C_VEL
LIN {X 0,Y 559.966,Z 544.225,A -85,B 0,C 180,E1 -2957.566,E2 -2957.566} C_VEL
LIN {X 0,Y 559.819,Z 555.924,A -85,B 0,C 180,E1 -2957.981,E2 -2957.981} C_VEL
LIN {X 0,Y 559.668,Z 567.814,A -85,B 0,C 180,E1 -2958.547,E2 -2958.547} C_VEL
LIN {X 0,Y 559.507,Z 578.909,A -85,B 0,C 180,E1 -2959.231,E2 -2959.231} C_VEL
LIN {X 0,Y 559.312,Z 589.541,A -85,B 0,C 180,E1 -2960.051,E2 -2960.051} C_VEL
LIN {X 0,Y 559.161,Z 599.114,A -85,B 0,C 180,E1 -2960.961,E2 -2960.961} C_VEL
LIN {X 0,Y 559.05,Z 606.962,A -85,B 0,C 180,E1 -2961.87,E2 -2961.87} C_VEL
LIN {X 0,Y 558.944,Z 614.623,A -85,B 0,C 180,E1 -2962.958,E2 -2962.958} C_VEL
LIN {X 0,Y 558.935,Z 621.68,A -85,B 0,C 180,E1 -2964.227,E2 -2964.227} C_VEL
LIN {X 0,Y 558.827,Z 626.373,A -85,B 0,C 180,E1 -2965.311,E2 -2965.311} C_VEL
LIN {X 0,Y 558.836,Z 629.958,A -85,B 0,C 180,E1 -2966.395,E2 -2966.395} C_VEL
LIN {X 0,Y 558.799,Z 631.808,A -85,B 0,C 180,E1 -2967.116,E2 -2967.116} C_VEL
LIN {X 0,Y 558.745,Z 634.184,A -85,B 0,C 180,E1 -2968.559,E2 -2968.559} C_VEL
LIN {X 0,Y 558.74,Z 635,A -85,B 0,C 180,E1 -2970,E2 -2970} C_VEL
LIN {X 0,Y 558.745,Z 634.185,A -85,B 0,C 180,E1 -2971.441,E2 -2971.441} C_VEL
LIN {X 0,Y 558.799,Z 631.81,A -85,B 0,C 180,E1 -2972.884,E2 -2972.884} C_VEL
LIN {X 0,Y 558.843,Z 628.896,A -85,B 0,C 180,E1 -2973.966,E2 -2973.966} C_VEL
LIN {X 0,Y 558.799,Z 624.949,A -85,B 0,C 180,E1 -2975.051,E2 -2975.051} C_VEL
LIN {X 0,Y 558.921,Z 619.868,A -85,B 0,C 180,E1 -2976.135,E2 -2976.135} C_VEL
LIN {X 0,Y 558.977,Z 613.469,A -85,B 0,C 180,E1 -2977.223,E2 -2977.223} C_VEL
LIN {X 0,Y 559.099,Z 605.479,A -85,B 0,C 180,E1 -2978.312,E2 -2978.312} C_VEL
LIN {X 0,Y 559.184,Z 597.336,A -85,B 0,C 180,E1 -2979.221,E2 -2979.221} C_VEL
LIN {X 0,Y 559.351,Z 587.402,A -85,B 0,C 180,E1 -2980.131,E2 -2980.131} C_VEL
LIN {X 0,Y 559.53,Z 576.368,A -85,B 0,C 180,E1 -2980.939,E2 -2980.939} C_VEL
LIN {X 0,Y 559.703,Z 564.145,A -85,B 0,C 180,E1 -2981.643,E2 -2981.643} C_VEL
LIN {X 0,Y 559.815,Z 551.774,A -85,B 0,C 180,E1 -2982.184,E2 -2982.184} C_VEL
LIN {X 0,Y 559.976,Z 538.355,A -85,B 0,C 180,E1 -2982.595,E2 -2982.595} C_VEL
LIN {X 0,Y 560.077,Z 525.101,A -85,B 0,C 180,E1 -2982.846,E2 -2982.846} C_VEL
LIN {X 0,Y 560.194,Z 425.623,A -85,B 0,C 180,E1 -2984.128,E2 -2984.128} C_VEL
LIN {X 0,Y 559.601,Z 420.911,A -85,B 0,C 180,E1 -2984.222,E2 -2984.222} C_VEL
LIN {X 0,Y 559.928,Z 393.758,A -85,B 0,C 180,E1 -2987.212,E2 -2987.212} C_VEL
LIN {X 0,Y 560.275,Z 368.924,A -85,B 0,C 180,E1 -2989.968,E2 -2989.968} C_VEL
LIN {X 0,Y 560.523,Z 344.149,A -85,B 0,C 180,E1 -2992.678,E2 -2992.678} C_VEL
LIN {X 0,Y 560.795,Z 318.436,A -85,B 0,C 180,E1 -2995.535,E2 -2995.535} C_VEL
LIN {X 0,Y 560.678,Z 308.864,A -85,B 0,C 180,E1 -2996.623,E2 -2996.623} C_VEL
LIN {X 0,Y 559.165,Z 301.944,A -85,B 0,C 180,E1 -2997.509,E2 -2997.509} C_VEL
LIN {X 0,Y 559.13,Z 301.833,A -85,B 0,C 180,E1 -3000.184,E2 -3000.184} C_VEL
LIN {X 0,Y 559.132,Z 301.832,A -85,B 0,C 180,E1 -3002.716,E2 -3002.716} C_VEL
LIN {X 0,Y 559.112,Z 301.835,A -85,B 0,C 180,E1 -3005.324,E2 -3005.324} C_VEL
LIN {X 0,Y 559.12,Z 301.842,A -85,B 0,C 180,E1 -3008.018,E2 -3008.018} C_VEL
LIN {X 0,Y 559.154,Z 301.834,A -85,B 0,C 180,E1 -3009.941,E2 -3009.941} C_VEL
LIN {X 0,Y 559.112,Z 301.835,A -85,B 0,C 180,E1 -3012.747,E2 -3012.747} C_VEL
LIN {X 0,Y 559.119,Z 301.834,A -85,B 0,C 180,E1 -3015.763,E2 -3015.763} C_VEL
LIN {X 0,Y 559.119,Z 301.839,A -85,B 0,C 180,E1 -3018.226,E2 -3018.226} C_VEL
LIN {X 0,Y 559.162,Z 301.825,A -85,B 0,C 180,E1 -3021.192,E2 -3021.192} C_VEL
LIN {X 0,Y 559.107,Z 301.831,A -85,B 0,C 180,E1 -3023.787,E2 -3023.787} C_VEL
LIN {X 0,Y 559.138,Z 301.832,A -85,B 0,C 180,E1 -3026.423,E2 -3026.423} C_VEL
LIN {X 0,Y 559.147,Z 301.83,A -85,B 0,C 180,E1 -3028.98,E2 -3028.98} C_VEL
LIN {X 0,Y 559.127,Z 301.836,A -85,B 0,C 180,E1 -3031.625,E2 -3031.625} C_VEL
LIN {X 0,Y 559.145,Z 301.839,A -85,B 0,C 180,E1 -3033.901,E2 -3033.901} C_VEL
LIN {X 0,Y 559.126,Z 301.832,A -85,B 0,C 180,E1 -3036.573,E2 -3036.573} C_VEL
LIN {X 0,Y 559.165,Z 301.826,A -85,B 0,C 180,E1 -3039.395,E2 -3039.395} C_VEL
LIN {X 0,Y 559.118,Z 301.839,A -85,B 0,C 180,E1 -3041.685,E2 -3041.685} C_VEL
LIN {X 0,Y 559.144,Z 301.837,A -85,B 0,C 180,E1 -3043.947,E2 -3043.947} C_VEL
LIN {X 0,Y 559.149,Z 301.83,A -85,B 0,C 180,E1 -3046.183,E2 -3046.183} C_VEL
LIN {X 0,Y 559.18,Z 301.826,A -85,B 0,C 180,E1 -3049.133,E2 -3049.133} C_VEL
LIN {X 0,Y 559.129,Z 301.835,A -85,B 0,C 180,E1 -3052.053,E2 -3052.053} C_VEL
LIN {X 0,Y 559.198,Z 301.824,A -85,B 0,C 180,E1 -3054.23,E2 -3054.23} C_VEL
LIN {X 0,Y 559.213,Z 301.823,A -85,B 0,C 180,E1 -3057.119,E2 -3057.119} C_VEL
LIN {X 0,Y 559.237,Z 301.82,A -85,B 0,C 180,E1 -3060,E2 -3060} C_VEL
LIN {X 0,Y 559.21,Z 301.821,A -85,B 0,C 180,E1 -3062.882,E2 -3062.882} C_VEL
LIN {X 0,Y 559.203,Z 301.829,A -85,B 0,C 180,E1 -3065.77,E2 -3065.77} C_VEL
LIN {X 0,Y 559.151,Z 301.827,A -85,B 0,C 180,E1 -3068.675,E2 -3068.675} C_VEL
LIN {X 0,Y 559.188,Z 301.834,A -85,B 0,C 180,E1 -3071.601,E2 -3071.601} C_VEL
LIN {X 0,Y 559.151,Z 301.826,A -85,B 0,C 180,E1 -3074.579,E2 -3074.579} C_VEL
LIN {X 0,Y 559.119,Z 301.843,A -85,B 0,C 180,E1 -3077.558,E2 -3077.558} C_VEL
LIN {X 0,Y 559.153,Z 301.832,A -85,B 0,C 180,E1 -3079.838,E2 -3079.838} C_VEL
LIN {X 0,Y 559.122,Z 301.834,A -85,B 0,C 180,E1 -3082.154,E2 -3082.154} C_VEL
LIN {X 0,Y 559.131,Z 301.836,A -85,B 0,C 180,E1 -3085.178,E2 -3085.178} C_VEL
LIN {X 0,Y 559.097,Z 301.836,A -85,B 0,C 180,E1 -3087.717,E2 -3087.717} C_VEL
LIN {X 0,Y 559.118,Z 301.827,A -85,B 0,C 180,E1 -3090.576,E2 -3090.576} C_VEL
LIN {X 0,Y 558.461,Z 301.915,A -85,B 0,C 180,E1 -3091.178,E2 -3091.178} C_VEL
LIN {X 0,Y 555.603,Z 302.27,A -85,B 0,C 180,E1 -3092.154,E2 -3092.154} C_VEL
LIN {X 0,Y 553.186,Z 302.572,A -85,B 0,C 180,E1 -3092.939,E2 -3092.939} C_VEL
LIN {X 0,Y 552.157,Z 302.71,A -85,B 0,C 180,E1 -3093.546,E2 -3093.546} C_VEL
LIN {X 0,Y 552.078,Z 302.711,A -85,B 0,C 180,E1 -3093.751,E2 -3093.751} C_VEL
LIN {X 0,Y 552.091,Z 302.708,A -85,B 0,C 180,E1 -3096.748,E2 -3096.748} C_VEL
LIN {X 0,Y 552.115,Z 302.708,A -85,B 0,C 180,E1 -3099.529,E2 -3099.529} C_VEL
LIN {X 0,Y 552.078,Z 302.71,A -85,B 0,C 180,E1 -3102.431,E2 -3102.431} C_VEL
LIN {X 0,Y 552.066,Z 302.715,A -85,B 0,C 180,E1 -3105.56,E2 -3105.56} C_VEL
LIN {X 0,Y 552.056,Z 302.712,A -85,B 0,C 180,E1 -3108.549,E2 -3108.549} C_VEL
LIN {X 0,Y 552.106,Z 302.713,A -85,B 0,C 180,E1 -3111.411,E2 -3111.411} C_VEL
LIN {X 0,Y 552.068,Z 302.712,A -85,B 0,C 180,E1 -3114.156,E2 -3114.156} C_VEL
LIN {X 0,Y 552.097,Z 302.714,A -85,B 0,C 180,E1 -3117.157,E2 -3117.157} C_VEL
LIN {X 0,Y 552.076,Z 302.712,A -85,B 0,C 180,E1 -3119.957,E2 -3119.957} C_VEL
LIN {X 0,Y 552.075,Z 302.709,A -85,B 0,C 180,E1 -3123.014,E2 -3123.014} C_VEL
LIN {X 0,Y 552.067,Z 302.714,A -85,B 0,C 180,E1 -3125.961,E2 -3125.961} C_VEL
LIN {X 0,Y 552.109,Z 302.705,A -85,B 0,C 180,E1 -3128.337,E2 -3128.337} C_VEL
LIN {X 0,Y 552.121,Z 302.708,A -85,B 0,C 180,E1 -3130.674,E2 -3130.674} C_VEL
LIN {X 0,Y 552.083,Z 302.704,A -85,B 0,C 180,E1 -3133.737,E2 -3133.737} C_VEL
LIN {X 0,Y 552.17,Z 302.917,A -85,B 0,C 180,E1 -3135.944,E2 -3135.944} C_VEL
LIN {X 0,Y 552.427,Z 304.035,A -85,B 0,C 180,E1 -3136.059,E2 -3136.059} C_VEL
LIN {X 0,Y 553.398,Z 307.022,A -85,B 0,C 180,E1 -3136.131,E2 -3136.131} C_VEL
LIN {X 0,Y 553.197,Z 382.292,A -85,B 0,C 180,E1 -3137.131,E2 -3137.131} C_VEL
LIN {X 0,Y 553.089,Z 395.472,A -85,B 0,C 180,E1 -3137.455,E2 -3137.455} C_VEL
LIN {X 0,Y 552.918,Z 407.533,A -85,B 0,C 180,E1 -3137.894,E2 -3137.894} C_VEL
LIN {X 0,Y 552.763,Z 418.912,A -85,B 0,C 180,E1 -3138.452,E2 -3138.452} C_VEL
LIN {X 0,Y 552.593,Z 430.429,A -85,B 0,C 180,E1 -3139.188,E2 -3139.188} C_VEL
LIN {X 0,Y 552.369,Z 440.793,A -85,B 0,C 180,E1 -3140.017,E2 -3140.017} C_VEL
LIN {X 0,Y 552.219,Z 449.24,A -85,B 0,C 180,E1 -3140.846,E2 -3140.846} C_VEL
LIN {X 0,Y 552.037,Z 457.012,A -85,B 0,C 180,E1 -3141.766,E2 -3141.766} C_VEL
LIN {X 0,Y 551.917,Z 464.7,A -85,B 0,C 180,E1 -3142.887,E2 -3142.887} C_VEL
LIN {X 0,Y 551.868,Z 471.526,A -85,B 0,C 180,E1 -3144.153,E2 -3144.153} C_VEL
LIN {X 0,Y 551.725,Z 476.199,A -85,B 0,C 180,E1 -3145.251,E2 -3145.251} C_VEL
LIN {X 0,Y 551.75,Z 479.829,A -85,B 0,C 180,E1 -3146.349,E2 -3146.349} C_VEL
LIN {X 0,Y 551.723,Z 481.708,A -85,B 0,C 180,E1 -3147.079,E2 -3147.079} C_VEL
LIN {X 0,Y 551.657,Z 483.128,A -85,B 0,C 180,E1 -3147.81,E2 -3147.81} C_VEL
LIN {X 0,Y 551.642,Z 484.756,A -85,B 0,C 180,E1 -3149.27,E2 -3149.27} C_VEL
LIN {X 0,Y 551.641,Z 484.996,A -85,B 0,C 180,E1 -3150,E2 -3150} C_VEL
LIN {X 0,Y 551.641,Z 484.815,A -85,B 0,C 180,E1 -3150.73,E2 -3150.73} C_VEL
LIN {X 0,Y 551.657,Z 483.266,A -85,B 0,C 180,E1 -3152.19,E2 -3152.19} C_VEL
LIN {X 0,Y 551.724,Z 481.905,A -85,B 0,C 180,E1 -3152.921,E2 -3152.921} C_VEL
LIN {X 0,Y 551.764,Z 479.025,A -85,B 0,C 180,E1 -3154.017,E2 -3154.017} C_VEL
LIN {X 0,Y 551.724,Z 475.129,A -85,B 0,C 180,E1 -3155.116,E2 -3155.116} C_VEL
LIN {X 0,Y 551.833,Z 469.521,A -85,B 0,C 180,E1 -3156.349,E2 -3156.349} C_VEL
LIN {X 0,Y 551.925,Z 462.823,A -85,B 0,C 180,E1 -3157.499,E2 -3157.499} C_VEL
LIN {X 0,Y 552.099,Z 454.806,A -85,B 0,C 180,E1 -3158.602,E2 -3158.602} C_VEL
LIN {X 0,Y 552.256,Z 446.593,A -85,B 0,C 180,E1 -3159.522,E2 -3159.522} C_VEL
LIN {X 0,Y 552.482,Z 436.435,A -85,B 0,C 180,E1 -3160.444,E2 -3160.444} C_VEL
LIN {X 0,Y 552.696,Z 425.859,A -85,B 0,C 180,E1 -3161.214,E2 -3161.214} C_VEL
LIN {X 0,Y 552.82,Z 415.483,A -85,B 0,C 180,E1 -3161.82,E2 -3161.82} C_VEL
LIN {X 0,Y 552.961,Z 404.093,A -85,B 0,C 180,E1 -3162.338,E2 -3162.338} C_VEL
LIN {X 0,Y 553.104,Z 391.349,A -85,B 0,C 180,E1 -3162.754,E2 -3162.754} C_VEL
LIN {X 0,Y 553.25,Z 379.266,A -85,B 0,C 180,E1 -3163.008,E2 -3163.008} C_VEL
LIN {X 0,Y 553.307,Z 306.752,A -85,B 0,C 180,E1 -3163.965,E2 -3163.965} C_VEL
LIN {X 0,Y 552.259,Z 303.528,A -85,B 0,C 180,E1 -3164.063,E2 -3164.063} C_VEL
LIN {X 0,Y 552.12,Z 302.744,A -85,B 0,C 180,E1 -3164.215,E2 -3164.215} C_VEL
LIN {X 0,Y 552.093,Z 302.681,A -85,B 0,C 180,E1 -3167.305,E2 -3167.305} C_VEL
LIN {X 0,Y 552.103,Z 302.709,A -85,B 0,C 180,E1 -3170.102,E2 -3170.102} C_VEL
LIN {X 0,Y 552.078,Z 302.712,A -85,B 0,C 180,E1 -3172.451,E2 -3172.451} C_VEL
LIN {X 0,Y 552.06,Z 302.714,A -85,B 0,C 180,E1 -3175.328,E2 -3175.328} C_VEL
LIN {X 0,Y 552.052,Z 302.708,A -85,B 0,C 180,E1 -3178.101,E2 -3178.101} C_VEL
LIN {X 0,Y 552.072,Z 302.718,A -85,B 0,C 180,E1 -3180.611,E2 -3180.611} C_VEL
LIN {X 0,Y 552.087,Z 302.712,A -85,B 0,C 180,E1 -3183.187,E2 -3183.187} C_VEL
LIN {X 0,Y 552.067,Z 302.712,A -85,B 0,C 180,E1 -3185.844,E2 -3185.844} C_VEL
LIN {X 0,Y 552.109,Z 302.711,A -85,B 0,C 180,E1 -3189.059,E2 -3189.059} C_VEL
LIN {X 0,Y 552.053,Z 302.713,A -85,B 0,C 180,E1 -3191.451,E2 -3191.451} C_VEL
LIN {X 0,Y 552.066,Z 302.715,A -85,B 0,C 180,E1 -3194.528,E2 -3194.528} C_VEL
LIN {X 0,Y 552.075,Z 302.711,A -85,B 0,C 180,E1 -3197.59,E2 -3197.59} C_VEL
LIN {X 0,Y 552.115,Z 302.709,A -85,B 0,C 180,E1 -3200.471,E2 -3200.471} C_VEL
LIN {X 0,Y 552.091,Z 302.708,A -85,B 0,C 180,E1 -3203.318,E2 -3203.318} C_VEL
LIN {X 0,Y 552.089,Z 302.71,A -85,B 0,C 180,E1 -3205.936,E2 -3205.936} C_VEL
LIN {X 0,Y 552.097,Z 302.711,A -85,B 0,C 180,E1 -3208.539,E2 -3208.539} C_VEL
LIN {X 0,Y 552.069,Z 302.704,A -85,B 0,C 180,E1 -3211.447,E2 -3211.447} C_VEL
LIN {X 0,Y 552.075,Z 302.716,A -85,B 0,C 180,E1 -3214.353,E2 -3214.353} C_VEL
LIN {X 0,Y 552.043,Z 302.72,A -85,B 0,C 180,E1 -3216.755,E2 -3216.755} C_VEL
LIN {X 0,Y 552.087,Z 302.708,A -85,B 0,C 180,E1 -3219.118,E2 -3219.118} C_VEL
LIN {X 0,Y 552.072,Z 302.711,A -85,B 0,C 180,E1 -3221.442,E2 -3221.442} C_VEL
LIN {X 0,Y 552.071,Z 302.711,A -85,B 0,C 180,E1 -3223.736,E2 -3223.736} C_VEL
LIN {X 0,Y 552.089,Z 302.708,A -85,B 0,C 180,E1 -3226.003,E2 -3226.003} C_VEL
LIN {X 0,Y 552.141,Z 302.704,A -85,B 0,C 180,E1 -3228.993,E2 -3228.993} C_VEL
LIN {X 0,Y 552.124,Z 302.705,A -85,B 0,C 180,E1 -3231.951,E2 -3231.951} C_VEL
LIN {X 0,Y 552.197,Z 302.698,A -85,B 0,C 180,E1 -3234.889,E2 -3234.889} C_VEL
LIN {X 0,Y 552.199,Z 302.696,A -85,B 0,C 180,E1 -3237.812,E2 -3237.812} C_VEL
LIN {X 0,Y 552.229,Z 302.695,A -85,B 0,C 180,E1 -3240.729,E2 -3240.729} C_VEL
LIN {X 0,Y 552.177,Z 302.699,A -85,B 0,C 180,E1 -3242.918,E2 -3242.918} C_VEL
LIN {X 0,Y 552.169,Z 302.699,A -85,B 0,C 180,E1 -3245.844,E2 -3245.844} C_VEL
LIN {X 0,Y 552.12,Z 302.708,A -85,B 0,C 180,E1 -3248.786,E2 -3248.786} C_VEL
LIN {X 0,Y 552.101,Z 302.709,A -85,B 0,C 180,E1 -3251.752,E2 -3251.752} C_VEL
LIN {X 0,Y 552.126,Z 302.707,A -85,B 0,C 180,E1 -3254.749,E2 -3254.749} C_VEL
LIN {X 0,Y 552.074,Z 302.714,A -85,B 0,C 180,E1 -3257.79,E2 -3257.79} C_VEL
LIN {X 0,Y 552.116,Z 302.71,A -85,B 0,C 180,E1 -3260.102,E2 -3260.102} C_VEL
LIN {X 0,Y 552.08,Z 302.715,A -85,B 0,C 180,E1 -3262.452,E2 -3262.452} C_VEL
LIN {X 0,Y 552.074,Z 302.711,A -85,B 0,C 180,E1 -3265.334,E2 -3265.334} C_VEL
LIN {X 0,Y 552.069,Z 302.717,A -85,B 0,C 180,E1 -3268.101,E2 -3268.101} C_VEL
LIN {X 0,Y 552.091,Z 302.712,A -85,B 0,C 180,E1 -3270.61,E2 -3270.61} C_VEL
LIN {X 0,Y 552.098,Z 302.707,A -85,B 0,C 180,E1 -3273.187,E2 -3273.187} C_VEL
LIN {X 0,Y 552.061,Z 302.716,A -85,B 0,C 180,E1 -3275.846,E2 -3275.846} C_VEL
LIN {X 0,Y 552.105,Z 302.708,A -85,B 0,C 180,E1 -3278.59,E2 -3278.59} C_VEL
LIN {X 0,Y 552.065,Z 302.714,A -85,B 0,C 180,E1 -3281.451,E2 -3281.451} C_VEL
LIN {X 0,Y 552.088,Z 302.71,A -85,B 0,C 180,E1 -3283.482,E2 -3283.482} C_VEL
LIN {X 0,Y 552.068,Z 302.714,A -85,B 0,C 180,E1 -3286.573,E2 -3286.573} C_VEL
LIN {X 0,Y 552.1,Z 302.713,A -85,B 0,C 180,E1 -3289.798,E2 -3289.798} C_VEL
LIN {X 0,Y 552.078,Z 302.716,A -85,B 0,C 180,E1 -3292.336,E2 -3292.336} C_VEL
LIN {X 0,Y 552.069,Z 302.712,A -85,B 0,C 180,E1 -3295.051,E2 -3295.051} C_VEL
LIN {X 0,Y 552.098,Z 302.712,A -85,B 0,C 180,E1 -3297.681,E2 -3297.681} C_VEL
LIN {X 0,Y 552.074,Z 302.705,A -85,B 0,C 180,E1 -3300.233,E2 -3300.233} C_VEL
LIN {X 0,Y 552.148,Z 302.895,A -85,B 0,C 180,E1 -3302.343,E2 -3302.343} C_VEL
LIN {X 0,Y 553.93,Z 311.551,A -85,B 0,C 180,E1 -3303.434,E2 -3303.434} C_VEL
LIN {X 0,Y 553.696,Z 335.522,A -85,B 0,C 180,E1 -3306.155,E2 -3306.155} C_VEL
LIN {X 0,Y 553.36,Z 362.577,A -85,B 0,C 180,E1 -3309.169,E2 -3309.169} C_VEL
LIN {X 0,Y 553.013,Z 390.621,A -85,B 0,C 180,E1 -3312.242,E2 -3312.242} C_VEL
LIN {X 0,Y 552.691,Z 414.777,A -85,B 0,C 180,E1 -3314.928,E2 -3314.928} C_VEL
LIN {X 0,Y 552.648,Z 420.912,A -85,B 0,C 180,E1 -3315.595,E2 -3315.595} C_VEL
LIN {X 0,Y 553.445,Z 428.527,A -85,B 0,C 180,E1 -3315.734,E2 -3315.734} C_VEL
LIN {X 0,Y 553.122,Z 530.957,A -85,B 0,C 180,E1 -3317.083,E2 -3317.083} C_VEL
LIN {X 0,Y 553.028,Z 544.224,A -85,B 0,C 180,E1 -3317.407,E2 -3317.407} C_VEL
LIN {X 0,Y 552.88,Z 556.375,A -85,B 0,C 180,E1 -3317.846,E2 -3317.846} C_VEL
LIN {X 0,Y 552.689,Z 568.672,A -85,B 0,C 180,E1 -3318.45,E2 -3318.45} C_VEL
LIN {X 0,Y 552.487,Z 580.198,A -85,B 0,C 180,E1 -3319.186,E2 -3319.186} C_VEL
LIN {X 0,Y 552.299,Z 590.607,A -85,B 0,C 180,E1 -3320.016,E2 -3320.016} C_VEL
LIN {X 0,Y 552.125,Z 599.115,A -85,B 0,C 180,E1 -3320.845,E2 -3320.845} C_VEL
LIN {X 0,Y 552.013,Z 606.962,A -85,B 0,C 180,E1 -3321.765,E2 -3321.765} C_VEL
LIN {X 0,Y 551.889,Z 614.622,A -85,B 0,C 180,E1 -3322.868,E2 -3322.868} C_VEL
LIN {X 0,Y 551.867,Z 621.68,A -85,B 0,C 180,E1 -3324.153,E2 -3324.153} C_VEL
LIN {X 0,Y 551.725,Z 626.373,A -85,B 0,C 180,E1 -3325.251,E2 -3325.251} C_VEL
LIN {X 0,Y 551.75,Z 629.958,A -85,B 0,C 180,E1 -3326.349,E2 -3326.349} C_VEL
LIN {X 0,Y 551.723,Z 631.807,A -85,B 0,C 180,E1 -3327.079,E2 -3327.079} C_VEL
LIN {X 0,Y 551.645,Z 634.184,A -85,B 0,C 180,E1 -3328.54,E2 -3328.54} C_VEL
LIN {X 0,Y 551.64,Z 635,A -85,B 0,C 180,E1 -3330,E2 -3330} C_VEL
LIN {X 0,Y 551.645,Z 634.185,A -85,B 0,C 180,E1 -3331.46,E2 -3331.46} C_VEL
LIN {X 0,Y 551.723,Z 631.81,A -85,B 0,C 180,E1 -3332.921,E2 -3332.921} C_VEL
LIN {X 0,Y 551.763,Z 628.896,A -85,B 0,C 180,E1 -3334.017,E2 -3334.017} C_VEL
LIN {X 0,Y 551.724,Z 624.949,A -85,B 0,C 180,E1 -3335.116,E2 -3335.116} C_VEL
LIN {X 0,Y 551.815,Z 619.124,A -85,B 0,C 180,E1 -3336.353,E2 -3336.353} C_VEL
LIN {X 0,Y 551.926,Z 612.237,A -85,B 0,C 180,E1 -3337.499,E2 -3337.499} C_VEL
LIN {X 0,Y 552.082,Z 603.993,A -85,B 0,C 180,E1 -3338.602,E2 -3338.602} C_VEL
LIN {X 0,Y 552.221,Z 595.541,A -85,B 0,C 180,E1 -3339.523,E2 -3339.523} C_VEL
LIN {X 0,Y 552.411,Z 585.096,A -85,B 0,C 180,E1 -3340.445,E2 -3340.445} C_VEL
LIN {X 0,Y 552.582,Z 574.131,A -85,B 0,C 180,E1 -3341.224,E2 -3341.224} C_VEL
LIN {X 0,Y 552.783,Z 563.41,A -85,B 0,C 180,E1 -3341.83,E2 -3341.83} C_VEL
LIN {X 0,Y 552.867,Z 551.77,A -85,B 0,C 180,E1 -3342.34,E2 -3342.34} C_VEL
LIN {X 0,Y 553.032,Z 539.269,A -85,B 0,C 180,E1 -3342.733,E2 -3342.733} C_VEL
LIN {X 0,Y 553.16,Z 526.616,A -85,B 0,C 180,E1 -3342.986,E2 -3342.986} C_VEL
LIN {X 0,Y 553.379,Z 426.74,A -85,B 0,C 180,E1 -3344.291,E2 -3344.291} C_VEL
LIN {X 0,Y 552.65,Z 420.918,A -85,B 0,C 180,E1 -3344.405,E2 -3344.405} C_VEL
LIN {X 0,Y 552.99,Z 393.204,A -85,B 0,C 180,E1 -3347.477,E2 -3347.477} C_VEL
LIN {X 0,Y 553.302,Z 366.088,A -85,B 0,C 180,E1 -3350.444,E2 -3350.444} C_VEL
LIN {X 0,Y 553.622,Z 339.74,A -85,B 0,C 180,E1 -3353.372,E2 -3353.372} C_VEL
LIN {X 0,Y 553.939,Z 314.952,A -85,B 0,C 180,E1 -3356.175,E2 -3356.175} C_VEL
LIN {X 0,Y 553.915,Z 311.549,A -85,B 0,C 180,E1 -3356.566,E2 -3356.566} C_VEL
LIN {X 0,Y 552.132,Z 302.823,A -85,B 0,C 180,E1 -3357.684,E2 -3357.684} C_VEL
LIN {X 0,Y 552.088,Z 302.712,A -85,B 0,C 180,E1 -3360.61,E2 -3360.61} C_VEL
LIN {X 0,Y 552.093,Z 302.708,A -85,B 0,C 180,E1 -3363.187,E2 -3363.187} C_VEL
LIN {X 0,Y 552.065,Z 302.717,A -85,B 0,C 180,E1 -3365.844,E2 -3365.844} C_VEL
LIN {X 0,Y 552.108,Z 302.707,A -85,B 0,C 180,E1 -3368.589,E2 -3368.589} C_VEL
LIN {X 0,Y 552.063,Z 302.714,A -85,B 0,C 180,E1 -3371.45,E2 -3371.45} C_VEL
LIN {X 0,Y 552.069,Z 302.706,A -85,B 0,C 180,E1 -3374.529,E2 -3374.529} C_VEL
LIN {X 0,Y 552.103,Z 302.71,A -85,B 0,C 180,E1 -3377.587,E2 -3377.587} C_VEL
LIN {X 0,Y 552.119,Z 302.704,A -85,B 0,C 180,E1 -3380.472,E2 -3380.472} C_VEL
LIN {X 0,Y 552.045,Z 302.704,A -85,B 0,C 180,E1 -3383.324,E2 -3383.324} C_VEL
LIN {X 0,Y 552.09,Z 302.715,A -85,B 0,C 180,E1 -3385.936,E2 -3385.936} C_VEL
LIN {X 0,Y 552.113,Z 302.707,A -85,B 0,C 180,E1 -3388.54,E2 -3388.54} C_VEL
LIN {X 0,Y 552.09,Z 302.709,A -85,B 0,C 180,E1 -3391.443,E2 -3391.443} C_VEL
LIN {X 0,Y 552.072,Z 302.714,A -85,B 0,C 180,E1 -3394.353,E2 -3394.353} C_VEL
LIN {X 0,Y 552.084,Z 302.708,A -85,B 0,C 180,E1 -3396.757,E2 -3396.757} C_VEL
LIN {X 0,Y 552.108,Z 302.702,A -85,B 0,C 180,E1 -3399.119,E2 -3399.119} C_VEL
LIN {X 0,Y 552.078,Z 302.711,A -85,B 0,C 180,E1 -3401.443,E2 -3401.443} C_VEL
LIN {X 0,Y 552.094,Z 302.717,A -85,B 0,C 180,E1 -3403.737,E2 -3403.737} C_VEL
LIN {X 0,Y 552.117,Z 302.708,A -85,B 0,C 180,E1 -3406.004,E2 -3406.004} C_VEL
LIN {X 0,Y 552.15,Z 302.701,A -85,B 0,C 180,E1 -3408.993,E2 -3408.993} C_VEL
LIN {X 0,Y 552.099,Z 302.712,A -85,B 0,C 180,E1 -3411.951,E2 -3411.951} C_VEL
LIN {X 0,Y 552.171,Z 302.7,A -85,B 0,C 180,E1 -3414.156,E2 -3414.156} C_VEL
LIN {X 0,Y 552.179,Z 302.699,A -85,B 0,C 180,E1 -3417.082,E2 -3417.082} C_VEL
LIN {X 0,Y 552.207,Z 302.695,A -85,B 0,C 180,E1 -3420,E2 -3420} C_VEL
LIN {X 0,Y 552.179,Z 302.697,A -85,B 0,C 180,E1 -3422.918,E2 -3422.918} C_VEL
LIN {X 0,Y 552.173,Z 302.703,A -85,B 0,C 180,E1 -3425.844,E2 -3425.844} C_VEL
LIN {X 0,Y 552.123,Z 302.702,A -85,B 0,C 180,E1 -3428.786,E2 -3428.786} C_VEL
LIN {X 0,Y 552.143,Z 302.709,A -85,B 0,C 180,E1 -3431.751,E2 -3431.751} C_VEL
LIN {X 0,Y 552.113,Z 302.702,A -85,B 0,C 180,E1 -3434.749,E2 -3434.749} C_VEL
LIN {X 0,Y 552.078,Z 302.717,A -85,B 0,C 180,E1 -3437.79,E2 -3437.79} C_VEL
LIN {X 0,Y 552.114,Z 302.705,A -85,B 0,C 180,E1 -3440.102,E2 -3440.102} C_VEL
LIN {X 0,Y 552.074,Z 302.71,A -85,B 0,C 180,E1 -3442.452,E2 -3442.452} C_VEL
LIN {X 0,Y 552.075,Z 302.717,A -85,B 0,C 180,E1 -3445.335,E2 -3445.335} C_VEL
LIN {X 0,Y 552.046,Z 302.709,A -85,B 0,C 180,E1 -3448.102,E2 -3448.102} C_VEL
LIN {X 0,Y 552.084,Z 302.702,A -85,B 0,C 180,E1 -3450.611,E2 -3450.611} C_VEL
LIN {X 0,Y 552.097,Z 302.711,A -85,B 0,C 180,E1 -3453.187,E2 -3453.187} C_VEL
LIN {X 0,Y 552.078,Z 302.711,A -85,B 0,C 180,E1 -3453.751,E2 -3453.751} C_VEL
LIN {X 0,Y 551.435,Z 302.794,A -85,B 0,C 180,E1 -3454.36,E2 -3454.36} C_VEL
LIN {X 0,Y 548.625,Z 303.148,A -85,B 0,C 180,E1 -3455.349,E2 -3455.349} C_VEL
LIN {X 0,Y 546.219,Z 303.442,A -85,B 0,C 180,E1 -3456.144,E2 -3456.144} C_VEL
LIN {X 0,Y 545.155,Z 303.573,A -85,B 0,C 180,E1 -3456.758,E2 -3456.758} C_VEL
LIN {X 0,Y 545.052,Z 303.587,A -85,B 0,C 180,E1 -3456.966,E2 -3456.966} C_VEL
LIN {X 0,Y 545.045,Z 303.583,A -85,B 0,C 180,E1 -3460.145,E2 -3460.145} C_VEL
LIN {X 0,Y 545.012,Z 303.595,A -85,B 0,C 180,E1 -3463.113,E2 -3463.113} C_VEL
LIN {X 0,Y 545.022,Z 303.585,A -85,B 0,C 180,E1 -3466.23,E2 -3466.23} C_VEL
LIN {X 0,Y 545.011,Z 303.592,A -85,B 0,C 180,E1 -3468.88,E2 -3468.88} C_VEL
LIN {X 0,Y 545.039,Z 303.588,A -85,B 0,C 180,E1 -3471.762,E2 -3471.762} C_VEL
LIN {X 0,Y 545.023,Z 303.589,A -85,B 0,C 180,E1 -3474.531,E2 -3474.531} C_VEL
LIN {X 0,Y 545.052,Z 303.592,A -85,B 0,C 180,E1 -3477.211,E2 -3477.211} C_VEL
LIN {X 0,Y 545.025,Z 303.592,A -85,B 0,C 180,E1 -3479.809,E2 -3479.809} C_VEL
LIN {X 0,Y 545.001,Z 303.584,A -85,B 0,C 180,E1 -3482.34,E2 -3482.34} C_VEL
LIN {X 0,Y 545.02,Z 303.592,A -85,B 0,C 180,E1 -3484.816,E2 -3484.816} C_VEL
LIN {X 0,Y 545.027,Z 303.592,A -85,B 0,C 180,E1 -3487.242,E2 -3487.242} C_VEL
LIN {X 0,Y 545.092,Z 303.582,A -85,B 0,C 180,E1 -3490.256,E2 -3490.256} C_VEL
LIN {X 0,Y 545.051,Z 303.571,A -85,B 0,C 180,E1 -3492.749,E2 -3492.749} C_VEL
LIN {X 0,Y 545.136,Z 303.771,A -85,B 0,C 180,E1 -3495.749,E2 -3495.749} C_VEL
LIN {X 0,Y 545.328,Z 304.687,A -85,B 0,C 180,E1 -3495.862,E2 -3495.862} C_VEL
LIN {X 0,Y 546.582,Z 308.927,A -85,B 0,C 180,E1 -3495.966,E2 -3495.966} C_VEL
LIN {X 0,Y 546.315,Z 383.303,A -85,B 0,C 180,E1 -3496.966,E2 -3496.966} C_VEL
LIN {X 0,Y 546.215,Z 396.461,A -85,B 0,C 180,E1 -3497.295,E2 -3497.295} C_VEL
LIN {X 0,Y 546.058,Z 408.171,A -85,B 0,C 180,E1 -3497.725,E2 -3497.725} C_VEL
LIN {X 0,Y 545.894,Z 419.957,A -85,B 0,C 180,E1 -3498.308,E2 -3498.308} C_VEL
LIN {X 0,Y 545.686,Z 431.415,A -85,B 0,C 180,E1 -3499.049,E2 -3499.049} C_VEL
LIN {X 0,Y 545.455,Z 441.774,A -85,B 0,C 180,E1 -3499.889,E2 -3499.889} C_VEL
LIN {X 0,Y 545.288,Z 450.221,A -85,B 0,C 180,E1 -3500.729,E2 -3500.729} C_VEL
LIN {X 0,Y 545.091,Z 457.991,A -85,B 0,C 180,E1 -3501.66,E2 -3501.66} C_VEL
LIN {X 0,Y 544.947,Z 465.683,A -85,B 0,C 180,E1 -3502.795,E2 -3502.795} C_VEL
LIN {X 0,Y 544.879,Z 472.506,A -85,B 0,C 180,E1 -3504.077,E2 -3504.077} C_VEL
LIN {X 0,Y 544.71,Z 477.139,A -85,B 0,C 180,E1 -3505.189,E2 -3505.189} C_VEL
LIN {X 0,Y 544.713,Z 480.666,A -85,B 0,C 180,E1 -3506.301,E2 -3506.301} C_VEL
LIN {X 0,Y 544.675,Z 482.495,A -85,B 0,C 180,E1 -3507.042,E2 -3507.042} C_VEL
LIN {X 0,Y 544.602,Z 483.882,A -85,B 0,C 180,E1 -3507.781,E2 -3507.781} C_VEL
LIN {X 0,Y 544.578,Z 485.464,A -85,B 0,C 180,E1 -3509.261,E2 -3509.261} C_VEL
LIN {X 0,Y 544.577,Z 485.698,A -85,B 0,C 180,E1 -3510,E2 -3510} C_VEL
LIN {X 0,Y 544.585,Z 484.954,A -85,B 0,C 180,E1 -3511.479,E2 -3511.479} C_VEL
LIN {X 0,Y 544.675,Z 482.683,A -85,B 0,C 180,E1 -3512.958,E2 -3512.958} C_VEL
LIN {X 0,Y 544.756,Z 479.876,A -85,B 0,C 180,E1 -3514.069,E2 -3514.069} C_VEL
LIN {X 0,Y 544.745,Z 476.087,A -85,B 0,C 180,E1 -3515.181,E2 -3515.181} C_VEL
LIN {X 0,Y 544.844,Z 470.89,A -85,B 0,C 180,E1 -3516.354,E2 -3516.354} C_VEL
LIN {X 0,Y 544.979,Z 463.795,A -85,B 0,C 180,E1 -3517.596,E2 -3517.596} C_VEL
LIN {X 0,Y 545.16,Z 455.781,A -85,B 0,C 180,E1 -3518.712,E2 -3518.712} C_VEL
LIN {X 0,Y 545.345,Z 447.565,A -85,B 0,C 180,E1 -3519.644,E2 -3519.644} C_VEL
LIN {X 0,Y 545.579,Z 438.551,A -85,B 0,C 180,E1 -3520.483,E2 -3520.483} C_VEL
LIN {X 0,Y 545.811,Z 428.112,A -85,B 0,C 180,E1 -3521.271,E2 -3521.271} C_VEL
LIN {X 0,Y 545.942,Z 416.451,A -85,B 0,C 180,E1 -3521.971,E2 -3521.971} C_VEL
LIN {X 0,Y 546.087,Z 405.062,A -85,B 0,C 180,E1 -3522.496,E2 -3522.496} C_VEL
LIN {X 0,Y 546.228,Z 392.301,A -85,B 0,C 180,E1 -3522.918,E2 -3522.918} C_VEL
LIN {X 0,Y 546.366,Z 380.207,A -85,B 0,C 180,E1 -3523.174,E2 -3523.174} C_VEL
LIN {X 0,Y 546.396,Z 307.92,A -85,B 0,C 180,E1 -3524.142,E2 -3524.142} C_VEL
LIN {X 0,Y 545.245,Z 304.457,A -85,B 0,C 180,E1 -3524.244,E2 -3524.244} C_VEL
LIN {X 0,Y 545.085,Z 303.639,A -85,B 0,C 180,E1 -3524.385,E2 -3524.385} C_VEL
LIN {X 0,Y 545.057,Z 303.556,A -85,B 0,C 180,E1 -3527.414,E2 -3527.414} C_VEL
LIN {X 0,Y 545.045,Z 303.591,A -85,B 0,C 180,E1 -3530.374,E2 -3530.374} C_VEL
LIN {X 0,Y 545.024,Z 303.591,A -85,B 0,C 180,E1 -3532.758,E2 -3532.758} C_VEL
LIN {X 0,Y 545.006,Z 303.591,A -85,B 0,C 180,E1 -3535.488,E2 -3535.488} C_VEL
LIN {X 0,Y 544.999,Z 303.584,A -85,B 0,C 180,E1 -3537.66,E2 -3537.66} C_VEL
LIN {X 0,Y 545.022,Z 303.591,A -85,B 0,C 180,E1 -3540.236,E2 -3540.236} C_VEL
LIN {X 0,Y 545.057,Z 303.589,A -85,B 0,C 180,E1 -3543.058,E2 -3543.058} C_VEL
LIN {X 0,Y 545.018,Z 303.59,A -85,B 0,C 180,E1 -3545.67,E2 -3545.67} C_VEL
LIN {X 0,Y 545.038,Z 303.587,A -85,B 0,C 180,E1 -3548.238,E2 -3548.238} C_VEL
LIN {X 0,Y 545.009,Z 303.593,A -85,B 0,C 180,E1 -3551.12,E2 -3551.12} C_VEL
LIN {X 0,Y 545.023,Z 303.587,A -85,B 0,C 180,E1 -3554.132,E2 -3554.132} C_VEL
LIN {X 0,Y 544.993,Z 303.599,A -85,B 0,C 180,E1 -3556.885,E2 -3556.885} C_VEL
LIN {X 0,Y 545.044,Z 303.583,A -85,B 0,C 180,E1 -3559.855,E2 -3559.855} C_VEL
LIN {X 0,Y 545.057,Z 303.587,A -85,B 0,C 180,E1 -3563.075,E2 -3563.075} C_VEL
LIN {X 0,Y 545.039,Z 303.593,A -85,B 0,C 180,E1 -3566.326,E2 -3566.326} C_VEL
LIN {X 0,Y 545.039,Z 303.583,A -85,B 0,C 180,E1 -3568.95,E2 -3568.95} C_VEL
LIN {X 0,Y 545.03,Z 303.58,A -85,B 0,C 180,E1 -3571.503,E2 -3571.503} C_VEL
LIN {X 0,Y 545.036,Z 303.587,A -85,B 0,C 180,E1 -3573.997,E2 -3573.997} C_VEL
LIN {X 0,Y 545.045,Z 303.595,A -85,B 0,C 180,E1 -3576.439,E2 -3576.439} C_VEL
LIN {X 0,Y 545.026,Z 303.591,A -85,B 0,C 180,E1 -3578.835,E2 -3578.835} C_VEL
LIN {X 0,Y 545.034,Z 303.588,A -85,B 0,C 180,E1 -3581.194,E2 -3581.194} C_VEL
LIN {X 0,Y 545.024,Z 303.588,A -85,B 0,C 180,E1 -3583.52,E2 -3583.52} C_VEL
LIN {X 0,Y 545.05,Z 303.583,A -85,B 0,C 180,E1 -3585.819,E2 -3585.819} C_VEL
LIN {X 0,Y 545.1,Z 303.583,A -85,B 0,C 180,E1 -3588.849,E2 -3588.849} C_VEL
LIN {X 0,Y 545.074,Z 303.582,A -85,B 0,C 180,E1 -3591.846,E2 -3591.846} C_VEL
LIN {X 0,Y 545.155,Z 303.576,A -85,B 0,C 180,E1 -3594.822,E2 -3594.822} C_VEL
LIN {X 0,Y 545.172,Z 303.571,A -85,B 0,C 180,E1 -3597.784,E2 -3597.784} C_VEL
LIN {X 0,Y 545.199,Z 303.57,A -85,B 0,C 180,E1 -3600.739,E2 -3600.739} C_VEL
LIN {X 0,Y 545.143,Z 303.575,A -85,B 0,C 180,E1 -3602.956,E2 -3602.956} C_VEL
LIN {X 0,Y 545.121,Z 303.578,A -85,B 0,C 180,E1 -3605.92,E2 -3605.92} C_VEL
LIN {X 0,Y 545.056,Z 303.591,A -85,B 0,C 180,E1 -3608.154,E2 -3608.154} C_VEL
LIN {X 0,Y 545.063,Z 303.583,A -85,B 0,C 180,E1 -3611.152,E2 -3611.152} C_VEL
LIN {X 0,Y 545.08,Z 303.588,A -85,B 0,C 180,E1 -3614.18,E2 -3614.18} C_VEL
LIN {X 0,Y 545.048,Z 303.586,A -85,B 0,C 180,E1 -3617.416,E2 -3617.416} C_VEL
LIN {X 0,Y 545.082,Z 303.583,A -85,B 0,C 180,E1 -3620.373,E2 -3620.373} C_VEL
LIN {X 0,Y 545.065,Z 303.584,A -85,B 0,C 180,E1 -3623.56,E2 -3623.56} C_VEL
LIN {X 0,Y 545.046,Z 303.585,A -85,B 0,C 180,E1 -3626.827,E2 -3626.827} C_VEL
LIN {X 0,Y 545.045,Z 303.584,A -85,B 0,C 180,E1 -3629.34,E2 -3629.34} C_VEL
LIN {X 0,Y 545.048,Z 303.592,A -85,B 0,C 180,E1 -3631.915,E2 -3631.915} C_VEL
LIN {X 0,Y 545.039,Z 303.588,A -85,B 0,C 180,E1 -3634.566,E2 -3634.566} C_VEL
LIN {X 0,Y 545.006,Z 303.592,A -85,B 0,C 180,E1 -3637.307,E2 -3637.307} C_VEL
LIN {X 0,Y 545.052,Z 303.594,A -85,B 0,C 180,E1 -3640.144,E2 -3640.144} C_VEL
LIN {X 0,Y 545.018,Z 303.588,A -85,B 0,C 180,E1 -3643.113,E2 -3643.113} C_VEL
LIN {X 0,Y 545.02,Z 303.596,A -85,B 0,C 180,E1 -3646.23,E2 -3646.23} C_VEL
LIN {X 0,Y 545.014,Z 303.59,A -85,B 0,C 180,E1 -3648.88,E2 -3648.88} C_VEL
LIN {X 0,Y 545.041,Z 303.591,A -85,B 0,C 180,E1 -3651.763,E2 -3651.763} C_VEL
LIN {X 0,Y 545.02,Z 303.592,A -85,B 0,C 180,E1 -3654.531,E2 -3654.531} C_VEL
LIN {X 0,Y 545.05,Z 303.585,A -85,B 0,C 180,E1 -3657.211,E2 -3657.211} C_VEL
LIN {X 0,Y 545.061,Z 303.582,A -85,B 0,C 180,E1 -3659.811,E2 -3659.811} C_VEL
LIN {X 0,Y 545.097,Z 303.774,A -85,B 0,C 180,E1 -3662.163,E2 -3662.163} C_VEL
LIN {X 0,Y 546.92,Z 312.425,A -85,B 0,C 180,E1 -3663.273,E2 -3663.273} C_VEL
LIN {X 0,Y 546.834,Z 326.529,A -85,B 0,C 180,E1 -3664.905,E2 -3664.905} C_VEL
LIN {X 0,Y 546.547,Z 350.312,A -85,B 0,C 180,E1 -3667.611,E2 -3667.611} C_VEL
LIN {X 0,Y 546.17,Z 375.666,A -85,B 0,C 180,E1 -3670.454,E2 -3670.454} C_VEL
LIN {X 0,Y 545.856,Z 401.924,A -85,B 0,C 180,E1 -3673.353,E2 -3673.353} C_VEL
LIN {X 0,Y 545.652,Z 420.816,A -85,B 0,C 180,E1 -3675.408,E2 -3675.408} C_VEL
LIN {X 0,Y 546.576,Z 428.52,A -85,B 0,C 180,E1 -3675.552,E2 -3675.552} C_VEL
LIN {X 0,Y 546.201,Z 530.957,A -85,B 0,C 180,E1 -3676.916,E2 -3676.916} C_VEL
LIN {X 0,Y 546.087,Z 544.224,A -85,B 0,C 180,E1 -3677.244,E2 -3677.244} C_VEL
LIN {X 0,Y 545.924,Z 556.374,A -85,B 0,C 180,E1 -3677.689,E2 -3677.689} C_VEL
LIN {X 0,Y 545.731,Z 568.67,A -85,B 0,C 180,E1 -3678.3,E2 -3678.3} C_VEL
LIN {X 0,Y 545.503,Z 580.196,A -85,B 0,C 180,E1 -3679.046,E2 -3679.046} C_VEL
LIN {X 0,Y 545.287,Z 590.607,A -85,B 0,C 180,E1 -3679.886,E2 -3679.886} C_VEL
LIN {X 0,Y 545.084,Z 599.115,A -85,B 0,C 180,E1 -3680.725,E2 -3680.725} C_VEL
LIN {X 0,Y 544.977,Z 606.962,A -85,B 0,C 180,E1 -3681.658,E2 -3681.658} C_VEL
LIN {X 0,Y 544.823,Z 614.622,A -85,B 0,C 180,E1 -3682.775,E2 -3682.775} C_VEL
LIN {X 0,Y 544.776,Z 621.68,A -85,B 0,C 180,E1 -3684.076,E2 -3684.076} C_VEL
LIN {X 0,Y 544.629,Z 626.373,A -85,B 0,C 180,E1 -3685.189,E2 -3685.189} C_VEL
LIN {X 0,Y 544.669,Z 629.958,A -85,B 0,C 180,E1 -3686.301,E2 -3686.301} C_VEL
LIN {X 0,Y 544.65,Z 631.807,A -85,B 0,C 180,E1 -3687.041,E2 -3687.041} C_VEL
LIN {X 0,Y 544.546,Z 634.183,A -85,B 0,C 180,E1 -3688.521,E2 -3688.521} C_VEL
LIN {X 0,Y 544.541,Z 635,A -85,B 0,C 180,E1 -3690,E2 -3690} C_VEL
LIN {X 0,Y 544.546,Z 634.184,A -85,B 0,C 180,E1 -3691.479,E2 -3691.479} C_VEL
LIN {X 0,Y 544.65,Z 631.81,A -85,B 0,C 180,E1 -3692.959,E2 -3692.959} C_VEL
LIN {X 0,Y 544.683,Z 628.896,A -85,B 0,C 180,E1 -3694.069,E2 -3694.069} C_VEL
LIN {X 0,Y 544.654,Z 624.949,A -85,B 0,C 180,E1 -3695.182,E2 -3695.182} C_VEL
LIN {X 0,Y 544.73,Z 619.643,A -85,B 0,C 180,E1 -3696.34,E2 -3696.34} C_VEL
LIN {X 0,Y 544.836,Z 613.468,A -85,B 0,C 180,E1 -3697.411,E2 -3697.411} C_VEL
LIN {X 0,Y 545.006,Z 605.478,A -85,B 0,C 180,E1 -3698.528,E2 -3698.528} C_VEL
LIN {X 0,Y 545.152,Z 597.335,A -85,B 0,C 180,E1 -3699.46,E2 -3699.46} C_VEL
LIN {X 0,Y 545.361,Z 587.399,A -85,B 0,C 180,E1 -3700.394,E2 -3700.394} C_VEL
LIN {X 0,Y 545.553,Z 576.54,A -85,B 0,C 180,E1 -3701.211,E2 -3701.211} C_VEL
LIN {X 0,Y 545.767,Z 565.175,A -85,B 0,C 180,E1 -3701.89,E2 -3701.89} C_VEL
LIN {X 0,Y 545.908,Z 552.977,A -85,B 0,C 180,E1 -3702.453,E2 -3702.453} C_VEL
LIN {X 0,Y 546.134,Z 540.182,A -85,B 0,C 180,E1 -3702.873,E2 -3702.873} C_VEL
LIN {X 0,Y 546.252,Z 526.615,A -85,B 0,C 180,E1 -3703.153,E2 -3703.153} C_VEL
LIN {X 0,Y 546.387,Z 426.659,A -85,B 0,C 180,E1 -3704.478,E2 -3704.478} C_VEL
LIN {X 0,Y 545.655,Z 420.809,A -85,B 0,C 180,E1 -3704.593,E2 -3704.593} C_VEL
LIN {X 0,Y 545.945,Z 393.141,A -85,B 0,C 180,E1 -3707.611,E2 -3707.611} C_VEL
LIN {X 0,Y 546.324,Z 365.185,A -85,B 0,C 180,E1 -3710.717,E2 -3710.717} C_VEL
LIN {X 0,Y 546.698,Z 339.124,A -85,B 0,C 180,E1 -3713.656,E2 -3713.656} C_VEL
LIN {X 0,Y 547.05,Z 314.209,A -85,B 0,C 180,E1 -3716.515,E2 -3716.515} C_VEL
LIN {X 0,Y 545.763,Z 306.965,A -85,B 0,C 180,E1 -3717.413,E2 -3717.413} C_VEL
LIN {X 0,Y 545.08,Z 303.703,A -85,B 0,C 180,E1 -3717.864,E2 -3717.864} C_VEL
LIN {X 0,Y 545.051,Z 303.587,A -85,B 0,C 180,E1 -3721.048,E2 -3721.048} C_VEL
LIN {X 0,Y 545.048,Z 303.59,A -85,B 0,C 180,E1 -3723.672,E2 -3723.672} C_VEL
LIN {X 0,Y 545.011,Z 303.596,A -85,B 0,C 180,E1 -3726.382,E2 -3726.382} C_VEL
LIN {X 0,Y 545.068,Z 303.583,A -85,B 0,C 180,E1 -3729.319,E2 -3729.319} C_VEL
LIN {X 0,Y 545.031,Z 303.596,A -85,B 0,C 180,E1 -3732.107,E2 -3732.107} C_VEL
LIN {X 0,Y 545.016,Z 303.583,A -85,B 0,C 180,E1 -3735.171,E2 -3735.171} C_VEL
LIN {X 0,Y 545.046,Z 303.595,A -85,B 0,C 180,E1 -3737.894,E2 -3737.894} C_VEL
LIN {X 0,Y 545.069,Z 303.58,A -85,B 0,C 180,E1 -3740.817,E2 -3740.817} C_VEL
LIN {X 0,Y 544.997,Z 303.583,A -85,B 0,C 180,E1 -3743.616,E2 -3743.616} C_VEL
LIN {X 0,Y 545.04,Z 303.59,A -85,B 0,C 180,E1 -3746.326,E2 -3746.326} C_VEL
LIN {X 0,Y 545.059,Z 303.585,A -85,B 0,C 180,E1 -3748.952,E2 -3748.952} C_VEL
LIN {X 0,Y 545.068,Z 303.584,A -85,B 0,C 180,E1 -3751.506,E2 -3751.506} C_VEL
LIN {X 0,Y 545.026,Z 303.59,A -85,B 0,C 180,E1 -3754.504,E2 -3754.504} C_VEL
LIN {X 0,Y 545.025,Z 303.59,A -85,B 0,C 180,E1 -3757.242,E2 -3757.242} C_VEL
LIN {X 0,Y 545.107,Z 303.577,A -85,B 0,C 180,E1 -3760.414,E2 -3760.414} C_VEL
LIN {X 0,Y 545.044,Z 303.592,A -85,B 0,C 180,E1 -3763.52,E2 -3763.52} C_VEL
LIN {X 0,Y 545.08,Z 303.588,A -85,B 0,C 180,E1 -3765.82,E2 -3765.82} C_VEL
LIN {X 0,Y 545.106,Z 303.578,A -85,B 0,C 180,E1 -3768.849,E2 -3768.849} C_VEL
LIN {X 0,Y 545.057,Z 303.591,A -85,B 0,C 180,E1 -3771.846,E2 -3771.846} C_VEL
LIN {X 0,Y 545.124,Z 303.578,A -85,B 0,C 180,E1 -3774.08,E2 -3774.08} C_VEL
LIN {X 0,Y 545.144,Z 303.575,A -85,B 0,C 180,E1 -3777.044,E2 -3777.044} C_VEL
LIN {X 0,Y 545.176,Z 303.571,A -85,B 0,C 180,E1 -3780,E2 -3780} C_VEL
LIN {X 0,Y 545.148,Z 303.573,A -85,B 0,C 180,E1 -3782.956,E2 -3782.956} C_VEL
LIN {X 0,Y 545.122,Z 303.58,A -85,B 0,C 180,E1 -3785.92,E2 -3785.92} C_VEL
LIN {X 0,Y 545.084,Z 303.579,A -85,B 0,C 180,E1 -3788.901,E2 -3788.901} C_VEL
LIN {X 0,Y 545.085,Z 303.586,A -85,B 0,C 180,E1 -3791.905,E2 -3791.905} C_VEL
LIN {X 0,Y 545.068,Z 303.581,A -85,B 0,C 180,E1 -3794.944,E2 -3794.944} C_VEL
LIN {X 0,Y 545.044,Z 303.589,A -85,B 0,C 180,E1 -3798.027,E2 -3798.027} C_VEL
LIN {X 0,Y 545.08,Z 303.579,A -85,B 0,C 180,E1 -3800.373,E2 -3800.373} C_VEL
LIN {X 0,Y 545.062,Z 303.594,A -85,B 0,C 180,E1 -3803.56,E2 -3803.56} C_VEL
LIN {X 0,Y 545.046,Z 303.585,A -85,B 0,C 180,E1 -3806.827,E2 -3806.827} C_VEL
LIN {X 0,Y 545.018,Z 303.588,A -85,B 0,C 180,E1 -3809.341,E2 -3809.341} C_VEL
LIN {X 0,Y 545.045,Z 303.588,A -85,B 0,C 180,E1 -3811.916,E2 -3811.916} C_VEL
LIN {X 0,Y 545.039,Z 303.587,A -85,B 0,C 180,E1 -3814.566,E2 -3814.566} C_VEL
LIN {X 0,Y 545.052,Z 303.587,A -85,B 0,C 180,E1 -3816.966,E2 -3816.966} C_VEL
LIN {X 0,Y 544.342,Z 303.68,A -85,B 0,C 180,E1 -3817.582,E2 -3817.582} C_VEL
LIN {X 0,Y 541.476,Z 304.037,A -85,B 0,C 180,E1 -3818.583,E2 -3818.583} C_VEL
LIN {X 0,Y 539.081,Z 304.33,A -85,B 0,C 180,E1 -3819.389,E2 -3819.389} C_VEL
LIN {X 0,Y 538.057,Z 304.455,A -85,B 0,C 180,E1 -3820.011,E2 -3820.011} C_VEL
LIN {X 0,Y 537.974,Z 304.463,A -85,B 0,C 180,E1 -3820.222,E2 -3820.222} C_VEL
LIN {X 0,Y 537.965,Z 304.471,A -85,B 0,C 180,E1 -3822.982,E2 -3822.982} C_VEL
LIN {X 0,Y 537.995,Z 304.462,A -85,B 0,C 180,E1 -3825.93,E2 -3825.93} C_VEL
LIN {X 0,Y 537.997,Z 304.471,A -85,B 0,C 180,E1 -3829.259,E2 -3829.259} C_VEL
LIN {X 0,Y 537.979,Z 304.464,A -85,B 0,C 180,E1 -3832.122,E2 -3832.122} C_VEL
LIN {X 0,Y 537.984,Z 304.469,A -85,B 0,C 180,E1 -3834.915,E2 -3834.915} C_VEL
LIN {X 0,Y 538.005,Z 304.468,A -85,B 0,C 180,E1 -3837.617,E2 -3837.617} C_VEL
LIN {X 0,Y 537.979,Z 304.467,A -85,B 0,C 180,E1 -3840.237,E2 -3840.237} C_VEL
LIN {X 0,Y 537.993,Z 304.459,A -85,B 0,C 180,E1 -3842.793,E2 -3842.793} C_VEL
LIN {X 0,Y 537.967,Z 304.478,A -85,B 0,C 180,E1 -3845.289,E2 -3845.289} C_VEL
LIN {X 0,Y 538.015,Z 304.461,A -85,B 0,C 180,E1 -3848.043,E2 -3848.043} C_VEL
LIN {X 0,Y 538.041,Z 304.46,A -85,B 0,C 180,E1 -3850.147,E2 -3850.147} C_VEL
LIN {X 0,Y 537.984,Z 304.449,A -85,B 0,C 180,E1 -3853.298,E2 -3853.298} C_VEL
LIN {X 0,Y 538.086,Z 304.612,A -85,B 0,C 180,E1 -3855.542,E2 -3855.542} C_VEL
LIN {X 0,Y 538.331,Z 305.686,A -85,B 0,C 180,E1 -3855.675,E2 -3855.675} C_VEL
LIN {X 0,Y 539.662,Z 309.635,A -85,B 0,C 180,E1 -3855.778,E2 -3855.778} C_VEL
LIN {X 0,Y 539.444,Z 384.313,A -85,B 0,C 180,E1 -3856.797,E2 -3856.797} C_VEL
LIN {X 0,Y 539.349,Z 397.459,A -85,B 0,C 180,E1 -3857.13,E2 -3857.13} C_VEL
LIN {X 0,Y 539.197,Z 410.388,A -85,B 0,C 180,E1 -3857.619,E2 -3857.619} C_VEL
LIN {X 0,Y 539.024,Z 422.111,A -85,B 0,C 180,E1 -3858.228,E2 -3858.228} C_VEL
LIN {X 0,Y 538.756,Z 433.671,A -85,B 0,C 180,E1 -3859.002,E2 -3859.002} C_VEL
LIN {X 0,Y 538.522,Z 443.806,A -85,B 0,C 180,E1 -3859.853,E2 -3859.853} C_VEL
LIN {X 0,Y 538.301,Z 452.886,A -85,B 0,C 180,E1 -3860.797,E2 -3860.797} C_VEL
LIN {X 0,Y 538.097,Z 461.669,A -85,B 0,C 180,E1 -3861.929,E2 -3861.929} C_VEL
LIN {X 0,Y 537.94,Z 467.863,A -85,B 0,C 180,E1 -3862.908,E2 -3862.908} C_VEL
LIN {X 0,Y 537.89,Z 473.485,A -85,B 0,C 180,E1 -3864,E2 -3864} C_VEL
LIN {X 0,Y 537.703,Z 478.118,A -85,B 0,C 180,E1 -3865.127,E2 -3865.127} C_VEL
LIN {X 0,Y 537.696,Z 481.646,A -85,B 0,C 180,E1 -3866.253,E2 -3866.253} C_VEL
LIN {X 0,Y 537.653,Z 483.474,A -85,B 0,C 180,E1 -3867.003,E2 -3867.003} C_VEL
LIN {X 0,Y 537.599,Z 484.858,A -85,B 0,C 180,E1 -3867.752,E2 -3867.752} C_VEL
LIN {X 0,Y 537.573,Z 486.44,A -85,B 0,C 180,E1 -3869.251,E2 -3869.251} C_VEL
LIN {X 0,Y 537.568,Z 486.674,A -85,B 0,C 180,E1 -3870,E2 -3870} C_VEL
LIN {X 0,Y 537.573,Z 486.496,A -85,B 0,C 180,E1 -3870.749,E2 -3870.749} C_VEL
LIN {X 0,Y 537.599,Z 484.986,A -85,B 0,C 180,E1 -3872.248,E2 -3872.248} C_VEL
LIN {X 0,Y 537.652,Z 483.659,A -85,B 0,C 180,E1 -3872.997,E2 -3872.997} C_VEL
LIN {X 0,Y 537.744,Z 480.854,A -85,B 0,C 180,E1 -3874.122,E2 -3874.122} C_VEL
LIN {X 0,Y 537.766,Z 477.061,A -85,B 0,C 180,E1 -3875.249,E2 -3875.249} C_VEL
LIN {X 0,Y 537.854,Z 471.894,A -85,B 0,C 180,E1 -3876.431,E2 -3876.431} C_VEL
LIN {X 0,Y 538.025,Z 464.766,A -85,B 0,C 180,E1 -3877.694,E2 -3877.694} C_VEL
LIN {X 0,Y 538.218,Z 456.754,A -85,B 0,C 180,E1 -3878.826,E2 -3878.826} C_VEL
LIN {X 0,Y 538.426,Z 448.538,A -85,B 0,C 180,E1 -3879.769,E2 -3879.769} C_VEL
LIN {X 0,Y 538.682,Z 439.519,A -85,B 0,C 180,E1 -3880.619,E2 -3880.619} C_VEL
LIN {X 0,Y 538.916,Z 429.064,A -85,B 0,C 180,E1 -3881.418,E2 -3881.418} C_VEL
LIN {X 0,Y 539.069,Z 417.418,A -85,B 0,C 180,E1 -3882.126,E2 -3882.126} C_VEL
LIN {X 0,Y 539.226,Z 406.026,A -85,B 0,C 180,E1 -3882.657,E2 -3882.657} C_VEL
LIN {X 0,Y 539.375,Z 393.257,A -85,B 0,C 180,E1 -3883.085,E2 -3883.085} C_VEL
LIN {X 0,Y 539.502,Z 381.151,A -85,B 0,C 180,E1 -3883.345,E2 -3883.345} C_VEL
LIN {X 0,Y 539.57,Z 309.422,A -85,B 0,C 180,E1 -3884.317,E2 -3884.317} C_VEL
LIN {X 0,Y 538.235,Z 305.45,A -85,B 0,C 180,E1 -3884.427,E2 -3884.427} C_VEL
LIN {X 0,Y 538.045,Z 304.523,A -85,B 0,C 180,E1 -3884.578,E2 -3884.578} C_VEL
LIN {X 0,Y 538.014,Z 304.432,A -85,B 0,C 180,E1 -3887.524,E2 -3887.524} C_VEL
LIN {X 0,Y 538.005,Z 304.472,A -85,B 0,C 180,E1 -3890.652,E2 -3890.652} C_VEL
LIN {X 0,Y 538.003,Z 304.468,A -85,B 0,C 180,E1 -3893.072,E2 -3893.072} C_VEL
LIN {X 0,Y 537.968,Z 304.467,A -85,B 0,C 180,E1 -3895.655,E2 -3895.655} C_VEL
LIN {X 0,Y 537.974,Z 304.46,A -85,B 0,C 180,E1 -3898.053,E2 -3898.053} C_VEL
LIN {X 0,Y 537.988,Z 304.473,A -85,B 0,C 180,E1 -3900.628,E2 -3900.628} C_VEL
LIN {X 0,Y 537.997,Z 304.466,A -85,B 0,C 180,E1 -3903.274,E2 -3903.274} C_VEL
LIN {X 0,Y 537.967,Z 304.469,A -85,B 0,C 180,E1 -3906.006,E2 -3906.006} C_VEL
LIN {X 0,Y 537.999,Z 304.472,A -85,B 0,C 180,E1 -3908.831,E2 -3908.831} C_VEL
LIN {X 0,Y 537.974,Z 304.466,A -85,B 0,C 180,E1 -3911.872,E2 -3911.872} C_VEL
LIN {X 0,Y 537.984,Z 304.472,A -85,B 0,C 180,E1 -3914.863,E2 -3914.863} C_VEL
LIN {X 0,Y 537.954,Z 304.472,A -85,B 0,C 180,E1 -3917.207,E2 -3917.207} C_VEL
LIN {X 0,Y 537.994,Z 304.464,A -85,B 0,C 180,E1 -3920.2,E2 -3920.2} C_VEL
LIN {X 0,Y 538.011,Z 304.464,A -85,B 0,C 180,E1 -3923.066,E2 -3923.066} C_VEL
LIN {X 0,Y 537.99,Z 304.466,A -85,B 0,C 180,E1 -3925.824,E2 -3925.824} C_VEL
LIN {X 0,Y 537.987,Z 304.468,A -85,B 0,C 180,E1 -3928.497,E2 -3928.497} C_VEL
LIN {X 0,Y 537.977,Z 304.46,A -85,B 0,C 180,E1 -3931.095,E2 -3931.095} C_VEL
LIN {X 0,Y 537.982,Z 304.464,A -85,B 0,C 180,E1 -3933.63,E2 -3933.63} C_VEL
LIN {X 0,Y 537.976,Z 304.471,A -85,B 0,C 180,E1 -3936.127,E2 -3936.127} C_VEL
LIN {X 0,Y 537.99,Z 304.47,A -85,B 0,C 180,E1 -3938.544,E2 -3938.544} C_VEL
LIN {X 0,Y 537.998,Z 304.467,A -85,B 0,C 180,E1 -3940.938,E2 -3940.938} C_VEL
LIN {X 0,Y 537.975,Z 304.467,A -85,B 0,C 180,E1 -3943.297,E2 -3943.297} C_VEL
LIN {X 0,Y 538.025,Z 304.457,A -85,B 0,C 180,E1 -3945.63,E2 -3945.63} C_VEL
LIN {X 0,Y 538.062,Z 304.461,A -85,B 0,C 180,E1 -3948.701,E2 -3948.701} C_VEL
LIN {X 0,Y 538.038,Z 304.457,A -85,B 0,C 180,E1 -3951.739,E2 -3951.739} C_VEL
LIN {X 0,Y 538.113,Z 304.454,A -85,B 0,C 180,E1 -3954.754,E2 -3954.754} C_VEL
LIN {X 0,Y 538.145,Z 304.446,A -85,B 0,C 180,E1 -3957.755,E2 -3957.755} C_VEL
LIN {X 0,Y 538.169,Z 304.446,A -85,B 0,C 180,E1 -3960.748,E2 -3960.748} C_VEL
LIN {X 0,Y 538.109,Z 304.451,A -85,B 0,C 180,E1 -3962.995,E2 -3962.995} C_VEL
LIN {X 0,Y 538.078,Z 304.456,A -85,B 0,C 180,E1 -3965.998,E2 -3965.998} C_VEL
LIN {X 0,Y 538.028,Z 304.468,A -85,B 0,C 180,E1 -3968.261,E2 -3968.261} C_VEL
LIN {X 0,Y 538.03,Z 304.46,A -85,B 0,C 180,E1 -3971.574,E2 -3971.574} C_VEL
LIN {X 0,Y 538.051,Z 304.459,A -85,B 0,C 180,E1 -3974.857,E2 -3974.857} C_VEL
LIN {X 0,Y 537.998,Z 304.47,A -85,B 0,C 180,E1 -3978.271,E2 -3978.271} C_VEL
LIN {X 0,Y 538.028,Z 304.458,A -85,B 0,C 180,E1 -3980.652,E2 -3980.652} C_VEL
LIN {X 0,Y 537.999,Z 304.468,A -85,B 0,C 180,E1 -3983.878,E2 -3983.878} C_VEL
LIN {X 0,Y 537.98,Z 304.471,A -85,B 0,C 180,E1 -3986.37,E2 -3986.37} C_VEL
LIN {X 0,Y 538.023,Z 304.458,A -85,B 0,C 180,E1 -3988.934,E2 -3988.934} C_VEL
LIN {X 0,Y 538.003,Z 304.47,A -85,B 0,C 180,E1 -3991.887,E2 -3991.887} C_VEL
LIN {X 0,Y 537.989,Z 304.466,A -85,B 0,C 180,E1 -3994.615,E2 -3994.615} C_VEL
LIN {X 0,Y 537.975,Z 304.474,A -85,B 0,C 180,E1 -3997.879,E2 -3997.879} C_VEL
LIN {X 0,Y 537.993,Z 304.466,A -85,B 0,C 180,E1 -4000.781,E2 -4000.781} C_VEL
LIN {X 0,Y 538.006,Z 304.464,A -85,B 0,C 180,E1 -4004.073,E2 -4004.073} C_VEL
LIN {X 0,Y 537.965,Z 304.468,A -85,B 0,C 180,E1 -4007.02,E2 -4007.02} C_VEL
LIN {X 0,Y 537.998,Z 304.464,A -85,B 0,C 180,E1 -4009.259,E2 -4009.259} C_VEL
LIN {X 0,Y 537.977,Z 304.476,A -85,B 0,C 180,E1 -4012.122,E2 -4012.122} C_VEL
LIN {X 0,Y 537.993,Z 304.467,A -85,B 0,C 180,E1 -4015.386,E2 -4015.386} C_VEL
LIN {X 0,Y 537.995,Z 304.474,A -85,B 0,C 180,E1 -4018.116,E2 -4018.116} C_VEL
LIN {X 0,Y 537.983,Z 304.458,A -85,B 0,C 180,E1 -4021.096,E2 -4021.096} C_VEL
LIN {X 0,Y 538.058,Z 304.727,A -85,B 0,C 180,E1 -4021.995,E2 -4021.995} C_VEL
LIN {X 0,Y 540.117,Z 315.086,A -85,B 0,C 180,E1 -4023.327,E2 -4023.327} C_VEL
LIN {X 0,Y 539.799,Z 338.557,A -85,B 0,C 180,E1 -4026.06,E2 -4026.06} C_VEL
LIN {X 0,Y 539.374,Z 364.293,A -85,B 0,C 180,E1 -4029.003,E2 -4029.003} C_VEL
LIN {X 0,Y 538.974,Z 391.302,A -85,B 0,C 180,E1 -4032.048,E2 -4032.048} C_VEL
LIN {X 0,Y 538.588,Z 419.288,A -85,B 0,C 180,E1 -4035.167,E2 -4035.167} C_VEL
LIN {X 0,Y 538.653,Z 420.77,A -85,B 0,C 180,E1 -4035.245,E2 -4035.245} C_VEL
LIN {X 0,Y 539.658,Z 429.8,A -85,B 0,C 180,E1 -4035.393,E2 -4035.393} C_VEL
LIN {X 0,Y 539.273,Z 530.284,A -85,B 0,C 180,E1 -4036.745,E2 -4036.745} C_VEL
LIN {X 0,Y 539.125,Z 543.65,A -85,B 0,C 180,E1 -4037.077,E2 -4037.077} C_VEL
LIN {X 0,Y 538.942,Z 557.063,A -85,B 0,C 180,E1 -4037.575,E2 -4037.575} C_VEL
LIN {X 0,Y 538.724,Z 569.099,A -85,B 0,C 180,E1 -4038.188,E2 -4038.188} C_VEL
LIN {X 0,Y 538.487,Z 581.407,A -85,B 0,C 180,E1 -4038.996,E2 -4038.996} C_VEL
LIN {X 0,Y 538.271,Z 591.646,A -85,B 0,C 180,E1 -4039.848,E2 -4039.848} C_VEL
LIN {X 0,Y 538.026,Z 600.787,A -85,B 0,C 180,E1 -4040.792,E2 -4040.792} C_VEL
LIN {X 0,Y 537.851,Z 609.688,A -85,B 0,C 180,E1 -4041.925,E2 -4041.925} C_VEL
LIN {X 0,Y 537.728,Z 616.849,A -85,B 0,C 180,E1 -4043.056,E2 -4043.056} C_VEL
LIN {X 0,Y 537.676,Z 623.366,A -85,B 0,C 180,E1 -4044.374,E2 -4044.374} C_VEL
LIN {X 0,Y 537.558,Z 627.677,A -85,B 0,C 180,E1 -4045.501,E2 -4045.501} C_VEL
LIN {X 0,Y 537.591,Z 629.958,A -85,B 0,C 180,E1 -4046.252,E2 -4046.252} C_VEL
LIN {X 0,Y 537.551,Z 631.807,A -85,B 0,C 180,E1 -4047.002,E2 -4047.002} C_VEL
LIN {X 0,Y 537.451,Z 634.182,A -85,B 0,C 180,E1 -4048.501,E2 -4048.501} C_VEL
LIN {X 0,Y 537.442,Z 635,A -85,B 0,C 180,E1 -4050,E2 -4050} C_VEL
LIN {X 0,Y 537.451,Z 634.184,A -85,B 0,C 180,E1 -4051.499,E2 -4051.499} C_VEL
LIN {X 0,Y 537.551,Z 631.81,A -85,B 0,C 180,E1 -4052.998,E2 -4052.998} C_VEL
LIN {X 0,Y 537.603,Z 628.895,A -85,B 0,C 180,E1 -4054.123,E2 -4054.123} C_VEL
LIN {X 0,Y 537.588,Z 624.948,A -85,B 0,C 180,E1 -4055.251,E2 -4055.251} C_VEL
LIN {X 0,Y 537.644,Z 620.125,A -85,B 0,C 180,E1 -4056.326,E2 -4056.326} C_VEL
LIN {X 0,Y 537.79,Z 613.467,A -85,B 0,C 180,E1 -4057.509,E2 -4057.509} C_VEL
LIN {X 0,Y 537.972,Z 605.478,A -85,B 0,C 180,E1 -4058.64,E2 -4058.64} C_VEL
LIN {X 0,Y 538.143,Z 597.334,A -85,B 0,C 180,E1 -4059.585,E2 -4059.585} C_VEL
LIN {X 0,Y 538.35,Z 587.379,A -85,B 0,C 180,E1 -4060.531,E2 -4060.531} C_VEL
LIN {X 0,Y 538.544,Z 577.454,A -85,B 0,C 180,E1 -4061.288,E2 -4061.288} C_VEL
LIN {X 0,Y 538.769,Z 566.736,A -85,B 0,C 180,E1 -4061.946,E2 -4061.946} C_VEL
LIN {X 0,Y 538.94,Z 553.631,A -85,B 0,C 180,E1 -4062.569,E2 -4062.569} C_VEL
LIN {X 0,Y 539.186,Z 540.493,A -85,B 0,C 180,E1 -4063.017,E2 -4063.017} C_VEL
LIN {X 0,Y 539.324,Z 527.428,A -85,B 0,C 180,E1 -4063.302,E2 -4063.302} C_VEL
LIN {X 0,Y 539.497,Z 427.357,A -85,B 0,C 180,E1 -4064.644,E2 -4064.644} C_VEL
LIN {X 0,Y 538.577,Z 419.803,A -85,B 0,C 180,E1 -4064.789,E2 -4064.789} C_VEL
LIN {X 0,Y 538.926,Z 394.53,A -85,B 0,C 180,E1 -4067.587,E2 -4067.587} C_VEL
LIN {X 0,Y 539.328,Z 366.04,A -85,B 0,C 180,E1 -4070.799,E2 -4070.799} C_VEL
LIN {X 0,Y 539.728,Z 341.489,A -85,B 0,C 180,E1 -4073.603,E2 -4073.603} C_VEL
LIN {X 0,Y 540.136,Z 316.842,A -85,B 0,C 180,E1 -4076.464,E2 -4076.464} C_VEL
LIN {X 0,Y 539.512,Z 311.473,A -85,B 0,C 180,E1 -4077.124,E2 -4077.124} C_VEL
LIN {X 0,Y 538.024,Z 304.628,A -85,B 0,C 180,E1 -4078.031,E2 -4078.031} C_VEL
LIN {X 0,Y 538,Z 304.468,A -85,B 0,C 180,E1 -4080.628,E2 -4080.628} C_VEL
LIN {X 0,Y 538.018,Z 304.462,A -85,B 0,C 180,E1 -4083.278,E2 -4083.278} C_VEL
LIN {X 0,Y 537.958,Z 304.474,A -85,B 0,C 180,E1 -4086.007,E2 -4086.007} C_VEL
LIN {X 0,Y 538.005,Z 304.462,A -85,B 0,C 180,E1 -4088.83,E2 -4088.83} C_VEL
LIN {X 0,Y 537.98,Z 304.475,A -85,B 0,C 180,E1 -4091.872,E2 -4091.872} C_VEL
LIN {X 0,Y 537.988,Z 304.457,A -85,B 0,C 180,E1 -4094.863,E2 -4094.863} C_VEL
LIN {X 0,Y 537.982,Z 304.466,A -85,B 0,C 180,E1 -4097.21,E2 -4097.21} C_VEL
LIN {X 0,Y 538.004,Z 304.462,A -85,B 0,C 180,E1 -4100.418,E2 -4100.418} C_VEL
LIN {X 0,Y 537.951,Z 304.455,A -85,B 0,C 180,E1 -4103.061,E2 -4103.061} C_VEL
LIN {X 0,Y 537.991,Z 304.468,A -85,B 0,C 180,E1 -4105.825,E2 -4105.825} C_VEL
LIN {X 0,Y 538.002,Z 304.465,A -85,B 0,C 180,E1 -4108.498,E2 -4108.498} C_VEL
LIN {X 0,Y 538.011,Z 304.459,A -85,B 0,C 180,E1 -4111.097,E2 -4111.097} C_VEL
LIN {X 0,Y 537.98,Z 304.47,A -85,B 0,C 180,E1 -4113.63,E2 -4113.63} C_VEL
LIN {X 0,Y 537.999,Z 304.468,A -85,B 0,C 180,E1 -4116.122,E2 -4116.122} C_VEL
LIN {X 0,Y 538.028,Z 304.457,A -85,B 0,C 180,E1 -4119.348,E2 -4119.348} C_VEL
LIN {X 0,Y 538.028,Z 304.461,A -85,B 0,C 180,E1 -4122.467,E2 -4122.467} C_VEL
LIN {X 0,Y 538.051,Z 304.465,A -85,B 0,C 180,E1 -4125.63,E2 -4125.63} C_VEL
LIN {X 0,Y 538.066,Z 304.455,A -85,B 0,C 180,E1 -4128.701,E2 -4128.701} C_VEL
LIN {X 0,Y 538.029,Z 304.468,A -85,B 0,C 180,E1 -4131.739,E2 -4131.739} C_VEL
LIN {X 0,Y 538.08,Z 304.457,A -85,B 0,C 180,E1 -4134.002,E2 -4134.002} C_VEL
LIN {X 0,Y 538.11,Z 304.451,A -85,B 0,C 180,E1 -4137.005,E2 -4137.005} C_VEL
LIN {X 0,Y 538.145,Z 304.446,A -85,B 0,C 180,E1 -4140,E2 -4140} C_VEL
LIN {X 0,Y 538.116,Z 304.45,A -85,B 0,C 180,E1 -4142.995,E2 -4142.995} C_VEL
LIN {X 0,Y 538.078,Z 304.456,A -85,B 0,C 180,E1 -4145.998,E2 -4145.998} C_VEL
LIN {X 0,Y 538.037,Z 304.458,A -85,B 0,C 180,E1 -4149.018,E2 -4149.018} C_VEL
LIN {X 0,Y 538.045,Z 304.461,A -85,B 0,C 180,E1 -4152.063,E2 -4152.063} C_VEL
LIN {X 0,Y 538.028,Z 304.459,A -85,B 0,C 180,E1 -4155.144,E2 -4155.144} C_VEL
LIN {X 0,Y 537.998,Z 304.465,A -85,B 0,C 180,E1 -4158.271,E2 -4158.271} C_VEL
LIN {X 0,Y 538.026,Z 304.458,A -85,B 0,C 180,E1 -4160.652,E2 -4160.652} C_VEL
LIN {X 0,Y 537.998,Z 304.469,A -85,B 0,C 180,E1 -4163.878,E2 -4163.878} C_VEL
LIN {X 0,Y 537.981,Z 304.464,A -85,B 0,C 180,E1 -4166.37,E2 -4166.37} C_VEL
LIN {X 0,Y 537.985,Z 304.459,A -85,B 0,C 180,E1 -4168.926,E2 -4168.926} C_VEL
LIN {X 0,Y 538.001,Z 304.465,A -85,B 0,C 180,E1 -4171.887,E2 -4171.887} C_VEL
LIN {X 0,Y 537.989,Z 304.466,A -85,B 0,C 180,E1 -4174.616,E2 -4174.616} C_VEL
LIN {X 0,Y 537.991,Z 304.469,A -85,B 0,C 180,E1 -4177.169,E2 -4177.169} C_VEL
LIN {X 0,Y 537.995,Z 304.464,A -85,B 0,C 180,E1 -4179.8,E2 -4179.8} C_VEL
LIN {X 0,Y 537.974,Z 304.463,A -85,B 0,C 180,E1 -4180.222,E2 -4180.222} C_VEL
LIN {X 0,Y 537.308,Z 304.547,A -85,B 0,C 180,E1 -4180.847,E2 -4180.847} C_VEL
LIN {X 0,Y 534.457,Z 304.914,A -85,B 0,C 180,E1 -4181.861,E2 -4181.861} C_VEL
LIN {X 0,Y 532.044,Z 305.22,A -85,B 0,C 180,E1 -4182.678,E2 -4182.678} C_VEL
LIN {X 0,Y 531.006,Z 305.346,A -85,B 0,C 180,E1 -4183.309,E2 -4183.309} C_VEL
LIN {X 0,Y 530.92,Z 305.354,A -85,B 0,C 180,E1 -4183.523,E2 -4183.523} C_VEL
LIN {X 0,Y 530.959,Z 305.341,A -85,B 0,C 180,E1 -4185.624,E2 -4185.624} C_VEL
LIN {X 0,Y 530.931,Z 305.347,A -85,B 0,C 180,E1 -4188.983,E2 -4188.983} C_VEL
LIN {X 0,Y 530.944,Z 305.346,A -85,B 0,C 180,E1 -4191.529,E2 -4191.529} C_VEL
LIN {X 0,Y 530.944,Z 305.343,A -85,B 0,C 180,E1 -4194.38,E2 -4194.38} C_VEL
LIN {X 0,Y 530.953,Z 305.348,A -85,B 0,C 180,E1 -4197.133,E2 -4197.133} C_VEL
LIN {X 0,Y 530.933,Z 305.347,A -85,B 0,C 180,E1 -4199.801,E2 -4199.801} C_VEL
LIN {X 0,Y 530.954,Z 305.333,A -85,B 0,C 180,E1 -4202.48,E2 -4202.48} C_VEL
LIN {X 0,Y 530.945,Z 305.347,A -85,B 0,C 180,E1 -4205.774,E2 -4205.774} C_VEL
LIN {X 0,Y 530.995,Z 305.341,A -85,B 0,C 180,E1 -4209.062,E2 -4209.062} C_VEL
LIN {X 0,Y 530.958,Z 305.331,A -85,B 0,C 180,E1 -4211.478,E2 -4211.478} C_VEL
LIN {X 0,Y 530.984,Z 305.345,A -85,B 0,C 180,E1 -4214.65,E2 -4214.65} C_VEL
LIN {X 0,Y 531.056,Z 305.597,A -85,B 0,C 180,E1 -4215.373,E2 -4215.373} C_VEL
LIN {X 0,Y 531.315,Z 306.677,A -85,B 0,C 180,E1 -4215.483,E2 -4215.483} C_VEL
LIN {X 0,Y 532.812,Z 311.037,A -85,B 0,C 180,E1 -4215.596,E2 -4215.596} C_VEL
LIN {X 0,Y 532.567,Z 385.325,A -85,B 0,C 180,E1 -4216.624,E2 -4216.624} C_VEL
LIN {X 0,Y 532.484,Z 398.459,A -85,B 0,C 180,E1 -4216.961,E2 -4216.961} C_VEL
LIN {X 0,Y 532.335,Z 411.38,A -85,B 0,C 180,E1 -4217.457,E2 -4217.457} C_VEL
LIN {X 0,Y 532.161,Z 422.253,A -85,B 0,C 180,E1 -4218.021,E2 -4218.021} C_VEL
LIN {X 0,Y 531.888,Z 433.387,A -85,B 0,C 180,E1 -4218.762,E2 -4218.762} C_VEL
LIN {X 0,Y 531.633,Z 443.741,A -85,B 0,C 180,E1 -4219.624,E2 -4219.624} C_VEL
LIN {X 0,Y 531.438,Z 452.183,A -85,B 0,C 180,E1 -4220.485,E2 -4220.485} C_VEL
LIN {X 0,Y 531.182,Z 459.955,A -85,B 0,C 180,E1 -4221.44,E2 -4221.44} C_VEL
LIN {X 0,Y 531.016,Z 467.645,A -85,B 0,C 180,E1 -4222.605,E2 -4222.605} C_VEL
LIN {X 0,Y 530.905,Z 474.465,A -85,B 0,C 180,E1 -4223.921,E2 -4223.921} C_VEL
LIN {X 0,Y 530.697,Z 479.098,A -85,B 0,C 180,E1 -4225.062,E2 -4225.062} C_VEL
LIN {X 0,Y 530.679,Z 482.626,A -85,B 0,C 180,E1 -4226.203,E2 -4226.203} C_VEL
LIN {X 0,Y 530.63,Z 484.454,A -85,B 0,C 180,E1 -4226.963,E2 -4226.963} C_VEL
LIN {X 0,Y 530.594,Z 485.834,A -85,B 0,C 180,E1 -4227.723,E2 -4227.723} C_VEL
LIN {X 0,Y 530.566,Z 487.415,A -85,B 0,C 180,E1 -4229.241,E2 -4229.241} C_VEL
LIN {X 0,Y 530.559,Z 487.649,A -85,B 0,C 180,E1 -4230,E2 -4230} C_VEL
LIN {X 0,Y 530.566,Z 487.47,A -85,B 0,C 180,E1 -4230.759,E2 -4230.759} C_VEL
LIN {X 0,Y 530.594,Z 485.96,A -85,B 0,C 180,E1 -4232.277,E2 -4232.277} C_VEL
LIN {X 0,Y 530.629,Z 484.636,A -85,B 0,C 180,E1 -4233.037,E2 -4233.037} C_VEL
LIN {X 0,Y 530.732,Z 481.83,A -85,B 0,C 180,E1 -4234.177,E2 -4234.177} C_VEL
LIN {X 0,Y 530.786,Z 478.034,A -85,B 0,C 180,E1 -4235.318,E2 -4235.318} C_VEL
LIN {X 0,Y 530.866,Z 472.891,A -85,B 0,C 180,E1 -4236.512,E2 -4236.512} C_VEL
LIN {X 0,Y 531.067,Z 465.739,A -85,B 0,C 180,E1 -4237.796,E2 -4237.796} C_VEL
LIN {X 0,Y 531.281,Z 457.727,A -85,B 0,C 180,E1 -4238.942,E2 -4238.942} C_VEL
LIN {X 0,Y 531.505,Z 449.51,A -85,B 0,C 180,E1 -4239.898,E2 -4239.898} C_VEL
LIN {X 0,Y 531.769,Z 440.491,A -85,B 0,C 180,E1 -4240.759,E2 -4240.759} C_VEL
LIN {X 0,Y 532.043,Z 430.032,A -85,B 0,C 180,E1 -4241.567,E2 -4241.567} C_VEL
LIN {X 0,Y 532.184,Z 418.541,A -85,B 0,C 180,E1 -4242.276,E2 -4242.276} C_VEL
LIN {X 0,Y 532.383,Z 406.028,A -85,B 0,C 180,E1 -4242.862,E2 -4242.862} C_VEL
LIN {X 0,Y 532.507,Z 393.307,A -85,B 0,C 180,E1 -4243.281,E2 -4243.281} C_VEL
LIN {X 0,Y 532.603,Z 382.1,A -85,B 0,C 180,E1 -4243.521,E2 -4243.521} C_VEL
LIN {X 0,Y 532.827,Z 311.207,A -85,B 0,C 180,E1 -4244.491,E2 -4244.491} C_VEL
LIN {X 0,Y 531.147,Z 306.172,A -85,B 0,C 180,E1 -4244.636,E2 -4244.636} C_VEL
LIN {X 0,Y 530.971,Z 305.385,A -85,B 0,C 180,E1 -4244.806,E2 -4244.806} C_VEL
LIN {X 0,Y 530.972,Z 305.309,A -85,B 0,C 180,E1 -4247.724,E2 -4247.724} C_VEL
LIN {X 0,Y 530.978,Z 305.344,A -85,B 0,C 180,E1 -4250.938,E2 -4250.938} C_VEL
LIN {X 0,Y 530.952,Z 305.343,A -85,B 0,C 180,E1 -4254.03,E2 -4254.03} C_VEL
LIN {X 0,Y 530.938,Z 305.341,A -85,B 0,C 180,E1 -4256.747,E2 -4256.747} C_VEL
LIN {X 0,Y 530.953,Z 305.344,A -85,B 0,C 180,E1 -4259.324,E2 -4259.324} C_VEL
LIN {X 0,Y 530.949,Z 305.343,A -85,B 0,C 180,E1 -4262.097,E2 -4262.097} C_VEL
LIN {X 0,Y 530.954,Z 305.35,A -85,B 0,C 180,E1 -4264.848,E2 -4264.848} C_VEL
LIN {X 0,Y 530.933,Z 305.341,A -85,B 0,C 180,E1 -4267.51,E2 -4267.51} C_VEL
LIN {X 0,Y 530.941,Z 305.349,A -85,B 0,C 180,E1 -4270.436,E2 -4270.436} C_VEL
LIN {X 0,Y 530.92,Z 305.34,A -85,B 0,C 180,E1 -4273.498,E2 -4273.498} C_VEL
LIN {X 0,Y 530.957,Z 305.341,A -85,B 0,C 180,E1 -4275.623,E2 -4275.623} C_VEL
LIN {X 0,Y 530.925,Z 305.345,A -85,B 0,C 180,E1 -4278.983,E2 -4278.983} C_VEL
LIN {X 0,Y 530.936,Z 305.337,A -85,B 0,C 180,E1 -4281.527,E2 -4281.527} C_VEL
LIN {X 0,Y 530.928,Z 305.35,A -85,B 0,C 180,E1 -4284.378,E2 -4284.378} C_VEL
LIN {X 0,Y 530.958,Z 305.341,A -85,B 0,C 180,E1 -4287.133,E2 -4287.133} C_VEL
LIN {X 0,Y 530.926,Z 305.336,A -85,B 0,C 180,E1 -4289.8,E2 -4289.8} C_VEL
LIN {X 0,Y 530.955,Z 305.341,A -85,B 0,C 180,E1 -4292.478,E2 -4292.478} C_VEL
LIN {X 0,Y 530.941,Z 305.347,A -85,B 0,C 180,E1 -4294.939,E2 -4294.939} C_VEL
LIN {X 0,Y 530.943,Z 305.348,A -85,B 0,C 180,E1 -4298.245,E2 -4298.245} C_VEL
LIN {X 0,Y 530.955,Z 305.348,A -85,B 0,C 180,E1 -4300.676,E2 -4300.676} C_VEL
LIN {X 0,Y 530.943,Z 305.344,A -85,B 0,C 180,E1 -4303.069,E2 -4303.069} C_VEL
LIN {X 0,Y 530.987,Z 305.333,A -85,B 0,C 180,E1 -4305.435,E2 -4305.435} C_VEL
LIN {X 0,Y 531.021,Z 305.341,A -85,B 0,C 180,E1 -4308.549,E2 -4308.549} C_VEL
LIN {X 0,Y 530.984,Z 305.335,A -85,B 0,C 180,E1 -4311.628,E2 -4311.628} C_VEL
LIN {X 0,Y 531.073,Z 305.332,A -85,B 0,C 180,E1 -4314.685,E2 -4314.685} C_VEL
LIN {X 0,Y 531.118,Z 305.321,A -85,B 0,C 180,E1 -4317.725,E2 -4317.725} C_VEL
LIN {X 0,Y 531.139,Z 305.321,A -85,B 0,C 180,E1 -4320.758,E2 -4320.758} C_VEL
LIN {X 0,Y 531.049,Z 305.33,A -85,B 0,C 180,E1 -4323.034,E2 -4323.034} C_VEL
LIN {X 0,Y 531.039,Z 305.334,A -85,B 0,C 180,E1 -4326.078,E2 -4326.078} C_VEL
LIN {X 0,Y 530.978,Z 305.347,A -85,B 0,C 180,E1 -4328.372,E2 -4328.372} C_VEL
LIN {X 0,Y 531.002,Z 305.336,A -85,B 0,C 180,E1 -4331.65,E2 -4331.65} C_VEL
LIN {X 0,Y 531.023,Z 305.334,A -85,B 0,C 180,E1 -4334.956,E2 -4334.956} C_VEL
LIN {X 0,Y 530.963,Z 305.343,A -85,B 0,C 180,E1 -4337.724,E2 -4337.724} C_VEL
LIN {X 0,Y 531.017,Z 305.335,A -85,B 0,C 180,E1 -4340.127,E2 -4340.127} C_VEL
LIN {X 0,Y 530.935,Z 305.347,A -85,B 0,C 180,E1 -4342.574,E2 -4342.574} C_VEL
LIN {X 0,Y 530.942,Z 305.344,A -85,B 0,C 180,E1 -4345.061,E2 -4345.061} C_VEL
LIN {X 0,Y 530.955,Z 305.341,A -85,B 0,C 180,E1 -4347.599,E2 -4347.599} C_VEL
LIN {X 0,Y 530.953,Z 305.349,A -85,B 0,C 180,E1 -4350.198,E2 -4350.198} C_VEL
LIN {X 0,Y 530.96,Z 305.341,A -85,B 0,C 180,E1 -4352.867,E2 -4352.867} C_VEL
LIN {X 0,Y 530.923,Z 305.346,A -85,B 0,C 180,E1 -4355.623,E2 -4355.623} C_VEL
LIN {X 0,Y 530.954,Z 305.341,A -85,B 0,C 180,E1 -4358.653,E2 -4358.653} C_VEL
LIN {X 0,Y 530.955,Z 305.344,A -85,B 0,C 180,E1 -4361.439,E2 -4361.439} C_VEL
LIN {X 0,Y 530.961,Z 305.334,A -85,B 0,C 180,E1 -4364.55,E2 -4364.55} C_VEL
LIN {X 0,Y 530.911,Z 305.35,A -85,B 0,C 180,E1 -4367.538,E2 -4367.538} C_VEL
LIN {X 0,Y 530.964,Z 305.34,A -85,B 0,C 180,E1 -4370.556,E2 -4370.556} C_VEL
LIN {X 0,Y 530.904,Z 305.351,A -85,B 0,C 180,E1 -4373.438,E2 -4373.438} C_VEL
LIN {X 0,Y 530.948,Z 305.347,A -85,B 0,C 180,E1 -4376.225,E2 -4376.225} C_VEL
LIN {X 0,Y 530.954,Z 305.345,A -85,B 0,C 180,E1 -4379.359,E2 -4379.359} C_VEL
LIN {X 0,Y 531.007,Z 305.521,A -85,B 0,C 180,E1 -4381.785,E2 -4381.785} C_VEL
LIN {X 0,Y 533.166,Z 315.949,A -85,B 0,C 180,E1 -4383.162,E2 -4383.162} C_VEL
LIN {X 0,Y 532.935,Z 335.662,A -85,B 0,C 180,E1 -4385.496,E2 -4385.496} C_VEL
LIN {X 0,Y 532.444,Z 361.646,A -85,B 0,C 180,E1 -4388.514,E2 -4388.514} C_VEL
LIN {X 0,Y 532.032,Z 386.085,A -85,B 0,C 180,E1 -4391.317,E2 -4391.317} C_VEL
LIN {X 0,Y 531.611,Z 412.166,A -85,B 0,C 180,E1 -4394.276,E2 -4394.276} C_VEL
LIN {X 0,Y 531.55,Z 418.82,A -85,B 0,C 180,E1 -4395.011,E2 -4395.011} C_VEL
LIN {X 0,Y 532.775,Z 430.155,A -85,B 0,C 180,E1 -4395.218,E2 -4395.218} C_VEL
LIN {X 0,Y 532.38,Z 529.298,A -85,B 0,C 180,E1 -4396.57,E2 -4396.57} C_VEL
LIN {X 0,Y 532.175,Z 542.658,A -85,B 0,C 180,E1 -4396.905,E2 -4396.905} C_VEL
LIN {X 0,Y 531.939,Z 556.064,A -85,B 0,C 180,E1 -4397.409,E2 -4397.409} C_VEL
LIN {X 0,Y 531.748,Z 567.13,A -85,B 0,C 180,E1 -4397.972,E2 -4397.972} C_VEL
LIN {X 0,Y 531.455,Z 579.103,A -85,B 0,C 180,E1 -4398.752,E2 -4398.752} C_VEL
LIN {X 0,Y 531.183,Z 589.703,A -85,B 0,C 180,E1 -4399.615,E2 -4399.615} C_VEL
LIN {X 0,Y 531.033,Z 598.4,A -85,B 0,C 180,E1 -4400.478,E2 -4400.478} C_VEL
LIN {X 0,Y 530.85,Z 606.432,A -85,B 0,C 180,E1 -4401.435,E2 -4401.435} C_VEL
LIN {X 0,Y 530.681,Z 614.292,A -85,B 0,C 180,E1 -4402.581,E2 -4402.581} C_VEL
LIN {X 0,Y 530.585,Z 621.542,A -85,B 0,C 180,E1 -4403.917,E2 -4403.917} C_VEL
LIN {X 0,Y 530.459,Z 626.319,A -85,B 0,C 180,E1 -4405.06,E2 -4405.06} C_VEL
LIN {X 0,Y 530.516,Z 629.947,A -85,B 0,C 180,E1 -4406.202,E2 -4406.202} C_VEL
LIN {X 0,Y 530.457,Z 631.804,A -85,B 0,C 180,E1 -4406.962,E2 -4406.962} C_VEL
LIN {X 0,Y 530.41,Z 633.192,A -85,B 0,C 180,E1 -4407.722,E2 -4407.722} C_VEL
LIN {X 0,Y 530.344,Z 634.785,A -85,B 0,C 180,E1 -4409.241,E2 -4409.241} C_VEL
LIN {X 0,Y 530.342,Z 635,A -85,B 0,C 180,E1 -4410,E2 -4410} C_VEL
LIN {X 0,Y 530.361,Z 634.183,A -85,B 0,C 180,E1 -4411.519,E2 -4411.519} C_VEL
LIN {X 0,Y 530.41,Z 633.195,A -85,B 0,C 180,E1 -4412.278,E2 -4412.278} C_VEL
LIN {X 0,Y 530.457,Z 631.807,A -85,B 0,C 180,E1 -4413.038,E2 -4413.038} C_VEL
LIN {X 0,Y 530.522,Z 628.876,A -85,B 0,C 180,E1 -4414.178,E2 -4414.178} C_VEL
LIN {X 0,Y 530.525,Z 624.876,A -85,B 0,C 180,E1 -4415.321,E2 -4415.321} C_VEL
LIN {X 0,Y 530.596,Z 619.075,A -85,B 0,C 180,E1 -4416.579,E2 -4416.579} C_VEL
LIN {X 0,Y 530.727,Z 611.841,A -85,B 0,C 180,E1 -4417.801,E2 -4417.801} C_VEL
LIN {X 0,Y 530.908,Z 603.395,A -85,B 0,C 180,E1 -4418.948,E2 -4418.948} C_VEL
LIN {X 0,Y 531.107,Z 594.749,A -85,B 0,C 180,E1 -4419.905,E2 -4419.905} C_VEL
LIN {X 0,Y 531.342,Z 584.089,A -85,B 0,C 180,E1 -4420.864,E2 -4420.864} C_VEL
LIN {X 0,Y 531.634,Z 572.953,A -85,B 0,C 180,E1 -4421.672,E2 -4421.672} C_VEL
LIN {X 0,Y 531.849,Z 562.063,A -85,B 0,C 180,E1 -4422.303,E2 -4422.303} C_VEL
LIN {X 0,Y 532.051,Z 550.274,A -85,B 0,C 180,E1 -4422.831,E2 -4422.831} C_VEL
LIN {X 0,Y 532.271,Z 536.74,A -85,B 0,C 180,E1 -4423.262,E2 -4423.262} C_VEL
LIN {X 0,Y 532.422,Z 523.406,A -85,B 0,C 180,E1 -4423.526,E2 -4423.526} C_VEL
LIN {X 0,Y 532.618,Z 427.94,A -85,B 0,C 180,E1 -4424.816,E2 -4424.816} C_VEL
LIN {X 0,Y 531.535,Z 418.844,A -85,B 0,C 180,E1 -4424.988,E2 -4424.988} C_VEL
LIN {X 0,Y 531.896,Z 393.422,A -85,B 0,C 180,E1 -4427.846,E2 -4427.846} C_VEL
LIN {X 0,Y 532.401,Z 365.149,A -85,B 0,C 180,E1 -4431.082,E2 -4431.082} C_VEL
LIN {X 0,Y 532.841,Z 338.839,A -85,B 0,C 180,E1 -4434.134,E2 -4434.134} C_VEL
LIN {X 0,Y 533.24,Z 317.715,A -85,B 0,C 180,E1 -4436.622,E2 -4436.622} C_VEL
LIN {X 0,Y 532.474,Z 312.335,A -85,B 0,C 180,E1 -4437.3,E2 -4437.3} C_VEL
LIN {X 0,Y 530.992,Z 305.453,A -85,B 0,C 180,E1 -4438.243,E2 -4438.243} C_VEL
LIN {X 0,Y 530.942,Z 305.345,A -85,B 0,C 180,E1 -4441.08,E2 -4441.08} C_VEL
LIN {X 0,Y 530.948,Z 305.347,A -85,B 0,C 180,E1 -4443.775,E2 -4443.775} C_VEL
LIN {X 0,Y 530.913,Z 305.35,A -85,B 0,C 180,E1 -4446.561,E2 -4446.561} C_VEL
LIN {X 0,Y 530.964,Z 305.34,A -85,B 0,C 180,E1 -4449.444,E2 -4449.444} C_VEL
LIN {X 0,Y 530.911,Z 305.35,A -85,B 0,C 180,E1 -4452.462,E2 -4452.462} C_VEL
LIN {X 0,Y 530.961,Z 305.334,A -85,B 0,C 180,E1 -4455.45,E2 -4455.45} C_VEL
LIN {X 0,Y 530.955,Z 305.344,A -85,B 0,C 180,E1 -4458.561,E2 -4458.561} C_VEL
LIN {X 0,Y 530.944,Z 305.342,A -85,B 0,C 180,E1 -4461.528,E2 -4461.528} C_VEL
LIN {X 0,Y 530.923,Z 305.342,A -85,B 0,C 180,E1 -4464.377,E2 -4464.377} C_VEL
LIN {X 0,Y 530.96,Z 305.341,A -85,B 0,C 180,E1 -4467.133,E2 -4467.133} C_VEL
LIN {X 0,Y 530.962,Z 305.348,A -85,B 0,C 180,E1 -4469.802,E2 -4469.802} C_VEL
LIN {X 0,Y 530.959,Z 305.34,A -85,B 0,C 180,E1 -4472.477,E2 -4472.477} C_VEL
LIN {X 0,Y 530.942,Z 305.344,A -85,B 0,C 180,E1 -4474.939,E2 -4474.939} C_VEL
LIN {X 0,Y 530.969,Z 305.341,A -85,B 0,C 180,E1 -4477.898,E2 -4477.898} C_VEL
LIN {X 0,Y 530.973,Z 305.336,A -85,B 0,C 180,E1 -4480.676,E2 -4480.676} C_VEL
LIN {X 0,Y 530.954,Z 305.342,A -85,B 0,C 180,E1 -4483.07,E2 -4483.07} C_VEL
LIN {X 0,Y 531.009,Z 305.339,A -85,B 0,C 180,E1 -4485.436,E2 -4485.436} C_VEL
LIN {X 0,Y 531.025,Z 305.332,A -85,B 0,C 180,E1 -4488.549,E2 -4488.549} C_VEL
LIN {X 0,Y 530.979,Z 305.347,A -85,B 0,C 180,E1 -4491.628,E2 -4491.628} C_VEL
LIN {X 0,Y 531.041,Z 305.335,A -85,B 0,C 180,E1 -4493.922,E2 -4493.922} C_VEL
LIN {X 0,Y 531.051,Z 305.33,A -85,B 0,C 180,E1 -4496.966,E2 -4496.966} C_VEL
LIN {X 0,Y 531.114,Z 305.322,A -85,B 0,C 180,E1 -4500,E2 -4500} C_VEL
LIN {X 0,Y 531.083,Z 305.326,A -85,B 0,C 180,E1 -4503.034,E2 -4503.034} C_VEL
LIN {X 0,Y 531.038,Z 305.332,A -85,B 0,C 180,E1 -4506.078,E2 -4506.078} C_VEL
LIN {X 0,Y 531,Z 305.335,A -85,B 0,C 180,E1 -4509.139,E2 -4509.139} C_VEL
LIN {X 0,Y 531.04,Z 305.339,A -85,B 0,C 180,E1 -4511.67,E2 -4511.67} C_VEL
LIN {X 0,Y 531.011,Z 305.331,A -85,B 0,C 180,E1 -4514.951,E2 -4514.951} C_VEL
LIN {X 0,Y 530.963,Z 305.348,A -85,B 0,C 180,E1 -4517.724,E2 -4517.724} C_VEL
LIN {X 0,Y 531.006,Z 305.334,A -85,B 0,C 180,E1 -4520.128,E2 -4520.128} C_VEL
LIN {X 0,Y 530.932,Z 305.344,A -85,B 0,C 180,E1 -4522.574,E2 -4522.574} C_VEL
LIN {X 0,Y 530.941,Z 305.346,A -85,B 0,C 180,E1 -4525.061,E2 -4525.061} C_VEL
LIN {X 0,Y 530.951,Z 305.341,A -85,B 0,C 180,E1 -4527.599,E2 -4527.599} C_VEL
LIN {X 0,Y 530.95,Z 305.332,A -85,B 0,C 180,E1 -4530.642,E2 -4530.642} C_VEL
LIN {X 0,Y 530.954,Z 305.349,A -85,B 0,C 180,E1 -4533.5,E2 -4533.5} C_VEL
LIN {X 0,Y 530.943,Z 305.342,A -85,B 0,C 180,E1 -4536.56,E2 -4536.56} C_VEL
LIN {X 0,Y 530.959,Z 305.34,A -85,B 0,C 180,E1 -4539.446,E2 -4539.446} C_VEL
LIN {X 0,Y 530.909,Z 305.347,A -85,B 0,C 180,E1 -4542.464,E2 -4542.464} C_VEL
LIN {X 0,Y 530.92,Z 305.354,A -85,B 0,C 180,E1 -4543.523,E2 -4543.523} C_VEL
LIN {X 0,Y 530.255,Z 305.432,A -85,B 0,C 180,E1 -4544.157,E2 -4544.157} C_VEL
LIN {X 0,Y 527.417,Z 305.788,A -85,B 0,C 180,E1 -4545.186,E2 -4545.186} C_VEL
LIN {X 0,Y 525.01,Z 306.081,A -85,B 0,C 180,E1 -4546.014,E2 -4546.014} C_VEL
LIN {X 0,Y 523.965,Z 306.208,A -85,B 0,C 180,E1 -4546.654,E2 -4546.654} C_VEL
LIN {X 0,Y 523.874,Z 306.219,A -85,B 0,C 180,E1 -4546.87,E2 -4546.87} C_VEL
LIN {X 0,Y 523.909,Z 306.222,A -85,B 0,C 180,E1 -4549.918,E2 -4549.918} C_VEL
LIN {X 0,Y 523.88,Z 306.221,A -85,B 0,C 180,E1 -4552.866,E2 -4552.866} C_VEL
LIN {X 0,Y 523.908,Z 306.223,A -85,B 0,C 180,E1 -4555.709,E2 -4555.709} C_VEL
LIN {X 0,Y 523.905,Z 306.22,A -85,B 0,C 180,E1 -4558.455,E2 -4558.455} C_VEL
LIN {X 0,Y 523.9,Z 306.225,A -85,B 0,C 180,E1 -4561.124,E2 -4561.124} C_VEL
LIN {X 0,Y 523.879,Z 306.224,A -85,B 0,C 180,E1 -4564.005,E2 -4564.005} C_VEL
LIN {X 0,Y 523.906,Z 306.221,A -85,B 0,C 180,E1 -4566.27,E2 -4566.27} C_VEL
LIN {X 0,Y 523.943,Z 306.215,A -85,B 0,C 180,E1 -4568.767,E2 -4568.767} C_VEL
LIN {X 0,Y 523.919,Z 306.211,A -85,B 0,C 180,E1 -4571.22,E2 -4571.22} C_VEL
LIN {X 0,Y 523.89,Z 306.203,A -85,B 0,C 180,E1 -4573.638,E2 -4573.638} C_VEL
LIN {X 0,Y 523.999,Z 306.435,A -85,B 0,C 180,E1 -4575.159,E2 -4575.159} C_VEL
LIN {X 0,Y 524.259,Z 307.528,A -85,B 0,C 180,E1 -4575.28,E2 -4575.28} C_VEL
LIN {X 0,Y 525.971,Z 312.481,A -85,B 0,C 180,E1 -4575.411,E2 -4575.411} C_VEL
LIN {X 0,Y 525.694,Z 386.337,A -85,B 0,C 180,E1 -4576.445,E2 -4576.445} C_VEL
LIN {X 0,Y 525.624,Z 399.458,A -85,B 0,C 180,E1 -4576.788,E2 -4576.788} C_VEL
LIN {X 0,Y 525.477,Z 412.372,A -85,B 0,C 180,E1 -4577.291,E2 -4577.291} C_VEL
LIN {X 0,Y 525.311,Z 422.9,A -85,B 0,C 180,E1 -4577.842,E2 -4577.842} C_VEL
LIN {X 0,Y 524.997,Z 434.372,A -85,B 0,C 180,E1 -4578.612,E2 -4578.612} C_VEL
LIN {X 0,Y 524.729,Z 444.725,A -85,B 0,C 180,E1 -4579.486,E2 -4579.486} C_VEL
LIN {X 0,Y 524.513,Z 453.166,A -85,B 0,C 180,E1 -4580.358,E2 -4580.358} C_VEL
LIN {X 0,Y 524.232,Z 460.938,A -85,B 0,C 180,E1 -4581.326,E2 -4581.326} C_VEL
LIN {X 0,Y 524.05,Z 468.626,A -85,B 0,C 180,E1 -4582.506,E2 -4582.506} C_VEL
LIN {X 0,Y 523.921,Z 475.445,A -85,B 0,C 180,E1 -4583.84,E2 -4583.84} C_VEL
LIN {X 0,Y 523.695,Z 480.079,A -85,B 0,C 180,E1 -4584.996,E2 -4584.996} C_VEL
LIN {X 0,Y 523.663,Z 483.606,A -85,B 0,C 180,E1 -4586.152,E2 -4586.152} C_VEL
LIN {X 0,Y 523.608,Z 485.434,A -85,B 0,C 180,E1 -4586.922,E2 -4586.922} C_VEL
LIN {X 0,Y 523.587,Z 486.811,A -85,B 0,C 180,E1 -4587.692,E2 -4587.692} C_VEL
LIN {X 0,Y 523.557,Z 488.391,A -85,B 0,C 180,E1 -4589.231,E2 -4589.231} C_VEL
LIN {X 0,Y 523.547,Z 488.625,A -85,B 0,C 180,E1 -4590,E2 -4590} C_VEL
LIN {X 0,Y 523.556,Z 488.445,A -85,B 0,C 180,E1 -4590.769,E2 -4590.769} C_VEL
LIN {X 0,Y 523.587,Z 486.935,A -85,B 0,C 180,E1 -4592.308,E2 -4592.308} C_VEL
LIN {X 0,Y 523.606,Z 485.613,A -85,B 0,C 180,E1 -4593.078,E2 -4593.078} C_VEL
LIN {X 0,Y 523.72,Z 482.807,A -85,B 0,C 180,E1 -4594.233,E2 -4594.233} C_VEL
LIN {X 0,Y 523.805,Z 479.008,A -85,B 0,C 180,E1 -4595.389,E2 -4595.389} C_VEL
LIN {X 0,Y 523.881,Z 473.882,A -85,B 0,C 180,E1 -4596.596,E2 -4596.596} C_VEL
LIN {X 0,Y 524.108,Z 466.713,A -85,B 0,C 180,E1 -4597.9,E2 -4597.9} C_VEL
LIN {X 0,Y 524.347,Z 458.699,A -85,B 0,C 180,E1 -4599.061,E2 -4599.061} C_VEL
LIN {X 0,Y 524.586,Z 450.482,A -85,B 0,C 180,E1 -4600.03,E2 -4600.03} C_VEL
LIN {X 0,Y 524.865,Z 441.462,A -85,B 0,C 180,E1 -4600.902,E2 -4600.902} C_VEL
LIN {X 0,Y 525.157,Z 430.993,A -85,B 0,C 180,E1 -4601.722,E2 -4601.722} C_VEL
LIN {X 0,Y 525.318,Z 419.508,A -85,B 0,C 180,E1 -4602.439,E2 -4602.439} C_VEL
LIN {X 0,Y 525.525,Z 406.991,A -85,B 0,C 180,E1 -4603.032,E2 -4603.032} C_VEL
LIN {X 0,Y 525.657,Z 394.263,A -85,B 0,C 180,E1 -4603.457,E2 -4603.457} C_VEL
LIN {X 0,Y 525.772,Z 381.542,A -85,B 0,C 180,E1 -4603.725,E2 -4603.725} C_VEL
LIN {X 0,Y 525.94,Z 312.407,A -85,B 0,C 180,E1 -4604.681,E2 -4604.681} C_VEL
LIN {X 0,Y 524.076,Z 306.994,A -85,B 0,C 180,E1 -4604.845,E2 -4604.845} C_VEL
LIN {X 0,Y 523.95,Z 306.309,A -85,B 0,C 180,E1 -4604.973,E2 -4604.973} C_VEL
LIN {X 0,Y 523.911,Z 306.19,A -85,B 0,C 180,E1 -4607.971,E2 -4607.971} C_VEL
LIN {X 0,Y 523.929,Z 306.222,A -85,B 0,C 180,E1 -4610.411,E2 -4610.411} C_VEL
LIN {X 0,Y 523.905,Z 306.221,A -85,B 0,C 180,E1 -4612.893,E2 -4612.893} C_VEL
LIN {X 0,Y 523.869,Z 306.225,A -85,B 0,C 180,E1 -4615.423,E2 -4615.423} C_VEL
LIN {X 0,Y 523.896,Z 306.211,A -85,B 0,C 180,E1 -4618.003,E2 -4618.003} C_VEL
LIN {X 0,Y 523.897,Z 306.228,A -85,B 0,C 180,E1 -4620.845,E2 -4620.845} C_VEL
LIN {X 0,Y 523.91,Z 306.219,A -85,B 0,C 180,E1 -4623.726,E2 -4623.726} C_VEL
LIN {X 0,Y 523.876,Z 306.228,A -85,B 0,C 180,E1 -4626.397,E2 -4626.397} C_VEL
LIN {X 0,Y 523.904,Z 306.224,A -85,B 0,C 180,E1 -4629.085,E2 -4629.085} C_VEL
LIN {X 0,Y 523.887,Z 306.223,A -85,B 0,C 180,E1 -4632.124,E2 -4632.124} C_VEL
LIN {X 0,Y 523.926,Z 306.218,A -85,B 0,C 180,E1 -4635.311,E2 -4635.311} C_VEL
LIN {X 0,Y 523.906,Z 306.223,A -85,B 0,C 180,E1 -4638.695,E2 -4638.695} C_VEL
LIN {X 0,Y 523.9,Z 306.213,A -85,B 0,C 180,E1 -4641.897,E2 -4641.897} C_VEL
LIN {X 0,Y 523.908,Z 306.224,A -85,B 0,C 180,E1 -4644.912,E2 -4644.912} C_VEL
LIN {X 0,Y 523.924,Z 306.215,A -85,B 0,C 180,E1 -4647.68,E2 -4647.68} C_VEL
LIN {X 0,Y 523.923,Z 306.211,A -85,B 0,C 180,E1 -4650.681,E2 -4650.681} C_VEL
LIN {X 0,Y 523.895,Z 306.219,A -85,B 0,C 180,E1 -4653.724,E2 -4653.724} C_VEL
LIN {X 0,Y 523.889,Z 306.228,A -85,B 0,C 180,E1 -4656.268,E2 -4656.268} C_VEL
LIN {X 0,Y 523.914,Z 306.22,A -85,B 0,C 180,E1 -4658.765,E2 -4658.765} C_VEL
LIN {X 0,Y 523.919,Z 306.219,A -85,B 0,C 180,E1 -4661.219,E2 -4661.219} C_VEL
LIN {X 0,Y 523.879,Z 306.223,A -85,B 0,C 180,E1 -4663.637,E2 -4663.637} C_VEL
LIN {X 0,Y 523.898,Z 306.219,A -85,B 0,C 180,E1 -4666.027,E2 -4666.027} C_VEL
LIN {X 0,Y 524.005,Z 306.216,A -85,B 0,C 180,E1 -4668.394,E2 -4668.394} C_VEL
LIN {X 0,Y 523.945,Z 306.212,A -85,B 0,C 180,E1 -4671.515,E2 -4671.515} C_VEL
LIN {X 0,Y 524.02,Z 306.212,A -85,B 0,C 180,E1 -4674.613,E2 -4674.613} C_VEL
LIN {X 0,Y 524.091,Z 306.197,A -85,B 0,C 180,E1 -4677.694,E2 -4677.694} C_VEL
LIN {X 0,Y 524.109,Z 306.197,A -85,B 0,C 180,E1 -4680.768,E2 -4680.768} C_VEL
LIN {X 0,Y 523.992,Z 306.209,A -85,B 0,C 180,E1 -4683.075,E2 -4683.075} C_VEL
LIN {X 0,Y 524.005,Z 306.211,A -85,B 0,C 180,E1 -4686.159,E2 -4686.159} C_VEL
LIN {X 0,Y 523.966,Z 306.212,A -85,B 0,C 180,E1 -4689.262,E2 -4689.262} C_VEL
LIN {X 0,Y 523.944,Z 306.218,A -85,B 0,C 180,E1 -4692.393,E2 -4692.393} C_VEL
LIN {X 0,Y 523.916,Z 306.219,A -85,B 0,C 180,E1 -4695.562,E2 -4695.562} C_VEL
LIN {X 0,Y 523.907,Z 306.225,A -85,B 0,C 180,E1 -4697.971,E2 -4697.971} C_VEL
LIN {X 0,Y 523.95,Z 306.212,A -85,B 0,C 180,E1 -4700.411,E2 -4700.411} C_VEL
LIN {X 0,Y 523.901,Z 306.22,A -85,B 0,C 180,E1 -4702.894,E2 -4702.894} C_VEL
LIN {X 0,Y 523.891,Z 306.222,A -85,B 0,C 180,E1 -4705.422,E2 -4705.422} C_VEL
LIN {X 0,Y 523.905,Z 306.223,A -85,B 0,C 180,E1 -4708.003,E2 -4708.003} C_VEL
LIN {X 0,Y 523.932,Z 306.218,A -85,B 0,C 180,E1 -4710.854,E2 -4710.854} C_VEL
LIN {X 0,Y 523.92,Z 306.221,A -85,B 0,C 180,E1 -4713.73,E2 -4713.73} C_VEL
LIN {X 0,Y 523.855,Z 306.232,A -85,B 0,C 180,E1 -4716.395,E2 -4716.395} C_VEL
LIN {X 0,Y 523.905,Z 306.217,A -85,B 0,C 180,E1 -4719.086,E2 -4719.086} C_VEL
LIN {X 0,Y 523.902,Z 306.227,A -85,B 0,C 180,E1 -4722.124,E2 -4722.124} C_VEL
LIN {X 0,Y 523.929,Z 306.207,A -85,B 0,C 180,E1 -4725.312,E2 -4725.312} C_VEL
LIN {X 0,Y 523.912,Z 306.22,A -85,B 0,C 180,E1 -4728.695,E2 -4728.695} C_VEL
LIN {X 0,Y 523.897,Z 306.226,A -85,B 0,C 180,E1 -4731.897,E2 -4731.897} C_VEL
LIN {X 0,Y 523.911,Z 306.22,A -85,B 0,C 180,E1 -4734.914,E2 -4734.914} C_VEL
LIN {X 0,Y 523.927,Z 306.22,A -85,B 0,C 180,E1 -4737.682,E2 -4737.682} C_VEL
LIN {X 0,Y 523.934,Z 306.203,A -85,B 0,C 180,E1 -4740.681,E2 -4740.681} C_VEL
LIN {X 0,Y 523.972,Z 306.469,A -85,B 0,C 180,E1 -4741.607,E2 -4741.607} C_VEL
LIN {X 0,Y 526.315,Z 318.036,A -85,B 0,C 180,E1 -4743.145,E2 -4743.145} C_VEL
LIN {X 0,Y 525.911,Z 341.468,A -85,B 0,C 180,E1 -4745.947,E2 -4745.947} C_VEL
